METHOD M_User_SetAction : INT
VAR_INPUT
END_VAR
// TODO USER
//
// This method implements the logic for controlling a heater.
// There are two input values from sensors and two deltas for comparison.
//
// This example implements the heater control with the following assumptions:
//
// in_lrTemp1 - Lowest Temperature in the system (L)
// in_lrTemp2 - Temperature of the Detector (D). Coming from Lakeshore.
//
// The heater should keep the System temperature  
// in_lrPar1 to in_lrPar2 lower than the detector temperature.
// 
// in_lrPar1  - Delta [K] to turn the heater ON:  IF L < D - in_lrPar1
// in_lrPar2  - Delta [K] to turn the heater OFF: IF L > D - in_lrPar2
//
// in_lrDelta1 > in_lrDelta2, e.g. 10K > 4K.
//
// For example:
// 	in_lrPar1 = 10K
// 	in_lrPar1 = 4K
// 	Detector temperature D = 100K
// 	The lowest system temperature is kept in range [(100-10)..(100-4)] = [90K..96K].
//	The heater is turned ON  at < 90K.
//	The heater is turned OFF at > 96K.
//
IF	stat.nState = E_CRYO_BIN_CTRL_STATE.ACTIVE_OFF  OR  
	stat.nState = E_CRYO_BIN_CTRL_STATE.ACTIVE_ON THEN
	
	IF in_lrTemp1 < in_lrTemp2 - in_lrDelta_Low THEN
		// Activate the actuator
		M_User_SetAction	:= E_CRYO_BIN_CTRL_ACTION.ON;
	ELSIF in_lrTemp1 > in_lrTemp2 - in_lrDelta_High THEN
		// Dectivate the actuator
		M_User_SetAction	:= E_CRYO_BIN_CTRL_ACTION.OFF;
	END_IF

ELSE
	// Don't do anything
	M_User_SetAction	:= E_CRYO_BIN_CTRL_ACTION.NONE;
END_IF
END_METHOD

END_FUNCTION_BLOCK

// POUs/Actuators/FB_CRYO_LN2_CTRL
FUNCTION_BLOCK FB_CRYO_LN2_CTRL EXTENDS FB_CRYO_BIN_CTRL
VAR_INPUT
	in_lrTempK:		LREAL;			// Temperature input value [K]
	in_bValid:		BOOL := TRUE;	// Temperature Valid flag
	// Two parameters for decision making
	in_lrTempValveOpen:		LREAL := 91.27;		// Open  valve if temperature above this value [K]
	in_lrTempValveClose:	LREAL := 79.148;	// Close valve if temperature below this value [K]
END_VAR
VAR_OUTPUT
END_VAR
VAR
END_VAR

// Check the validity of the temperature reading.
// Start the check after 200 cycles.
IF stat.nCycleCounter > 200 THEN
	IF NOT in_bValid THEN
		// The temperature is not valid. 
		// The controller cannot work.
		stat.bCtrlOK	:= FALSE;
	ELSIF in_lrTempValveClose >= in_lrTempValveOpen THEN
		// Wrong configuration.
		// ValveClose MUST be lower than ValveOpen temperature
		stat.bCtrlOK	:= FALSE;
	ELSE
		// The temperature is valid. 
		stat.bCtrlOK	:= TRUE;
	END_IF
ELSE
	// The temperature is valid. 
	stat.bCtrlOK	:= TRUE;
END_IF

// Execute parent FB.
SUPER^();

METHOD M_SetStatus
VAR_INPUT
	nState:	E_CRYO_BIN_CTRL_STATE;
END_VAR
// Execute the status of the parent FB
SUPER^.M_SetStatus(nState);

// Set proper error description, if any.
IF Actuator.stat.bError THEN
	stat.sState	:= 'Valve failure';
ELSIF NOT stat.bCtrlOK THEN
	stat.sState	:= 'Temperature not valid';
END_IF
END_METHOD

METHOD M_User_SetAction : INT
VAR_INPUT
END_VAR
// TODO USER
// Overwrite Method FB_CRYO_BIN_CTRL::M_User_SetOutput()
//
// This method implements the logic for controlling the LN2 valve.
// 
// FB_CRYO_LN2_CTRL input parameters:
//
// in_lrTempK          - LN2 temperature
// in_bValid           - Flag if temperature reading is valid
// in_lrTempValveOpen  - Temperature upper limit [K]. Valve opens  when:  LN2 > in_lrTempValveOpen
// in_lrTempValveClose - Temperature lower limit [K]. Valve closes when:  LN2 < in_lrTempValveClose
//
// in_lrTempValveOpen > in_lrTempValveClose, e.g. 91.27K > 79.148K.
//
	
IF	stat.nState = E_CRYO_BIN_CTRL_STATE.ACTIVE_OFF  OR  
	stat.nState = E_CRYO_BIN_CTRL_STATE.ACTIVE_ON THEN
	// Check if input temperature value is valid.
	// If OK, check temperature against the limits	
	IF NOT stat.bCtrlOK THEN
		// Temperature reading is not valid.
		// Dectivate the actuator, i.e. close the valve
		M_User_SetAction	:= E_CRYO_BIN_CTRL_ACTION.OFF;
		stat.nState	:= E_CRYO_BIN_CTRL_STATE.ERROR;
	ELSIF in_lrTempK > in_lrTempValveOpen THEN
		// Activate the actuator, i.e. open the valve
		M_User_SetAction	:= E_CRYO_BIN_CTRL_ACTION.ON;
	ELSIF in_lrTempK < in_lrTempValveClose THEN
		// Dectivate the actuator, i.e. close the valve
		M_User_SetAction	:= E_CRYO_BIN_CTRL_ACTION.OFF;
	END_IF
	
ELSE
	// Don't do anything
	M_User_SetAction	:= E_CRYO_BIN_CTRL_ACTION.NONE;
END_IF
END_METHOD

END_FUNCTION_BLOCK

// POUs/Actuators/FB_CRYO_VALVE_CTRL
FUNCTION_BLOCK FB_CRYO_VALVE_CTRL EXTENDS FB_CRYO_BIN_CTRL
VAR_INPUT
END_VAR
VAR_OUTPUT
END_VAR
VAR
END_VAR

// Execute parent FB.
SUPER^();

METHOD M_SetStatus
VAR_INPUT
	nState:	E_CRYO_BIN_CTRL_STATE;
END_VAR
// Execute the status of the parent FB
SUPER^.M_SetStatus(nState);

// Set proper error description, if any.
IF Actuator.stat.bError THEN
	stat.sState	:= 'Valve failure';
END_IF
END_METHOD

METHOD M_User_SetAction : INT
VAR_INPUT
END_VAR
// TODO USER
// Set Valve command based on the input parameter in_bEnable.
//
	
IF	stat.nState = E_CRYO_BIN_CTRL_STATE.ACTIVE_OFF  AND in_bEnable THEN
	// Activate the actuator, i.e. open the valve
	M_User_SetAction	:= E_CRYO_BIN_CTRL_ACTION.ON;
ELSIF  stat.nState = E_CRYO_BIN_CTRL_STATE.ACTIVE_ON AND NOT in_bEnable THEN
	// Dectivate the actuator, i.e. close the valve
	M_User_SetAction	:= E_CRYO_BIN_CTRL_ACTION.OFF;
ELSE
	// Don't do anything
	M_User_SetAction	:= E_CRYO_BIN_CTRL_ACTION.NONE;
END_IF
END_METHOD

END_FUNCTION_BLOCK

// POUs/Comm/FB_MODBUS_COMM_CPA
FUNCTION_BLOCK FB_MODBUS_COMM_CPA EXTENDS FB_MODBUS_COMM_BASE
VAR_INPUT
END_VAR
VAR_OUTPUT
END_VAR
VAR CONSTANT
END_VAR
VAR
	{attribute 'OPC.UA.DA' := '0'}
	sim:		FB_SIM_MODBUS_COMM_CPA;	// Reference to COMM simulator

END_VAR

simRef	REF=sim;

// Execute base FB, i.e. FB_MODBUS_COMM_BASE.
SUPER^();

END_FUNCTION_BLOCK

// POUs/Simulation/FB_SIM_MODBUS_COMM_CPA
FUNCTION_BLOCK FB_SIM_MODBUS_COMM_CPA EXTENDS FB_SIM_MODBUS_COMM_BASE
VAR_INPUT
END_VAR
VAR_OUTPUT
END_VAR
VAR
END_VAR

M_ActivityDo();

METHOD M_GetSimReply : STRING(255)
VAR_INPUT
	{attribute 'OPC.UA.DA' := '0'}
	cmd:	STRING(16);		// MODBUS command. Only first 8 bytes are used
END_VAR
VAR
	sReply:		ARRAY [0..300] OF BYTE;
	sReply1:	STRING(255);
	n2Bytes:	ARRAY [0..1] OF BYTE;	// 2 bytes
	n4Bytes:	ARRAY [0..3] OF BYTE;	// 4 bytes
	i:			INT;
	nRegister:	INT;
	nWords:		INT;
	nPos:		INT;	
END_VAR
// TODO User: Implement simulator replies in FBs that EXTEND FB_SIM_MODBUS_COMM_BASE.
//            Only case where cmd[1] = E_MODBUS_CMD_TYPE.READ should be implemented.

IF cmd[1] = E_MODBUS_CMD_TYPE.WRITE THEN
// This is a WRITE command.
// Reply is the same as the command.
(*
	FOR i:=0 TO 8 DO
		sReply[i]	:= cmd[i];
	END_FOR
	*)
	M_GetSimReply := cmd;	
ELSE
// This is a READ command
	// Get register number - cmd[2..3] swapped bytes
	nRegister	:= M_ByteSwapINT(ADR(cmd[2]));

	// Get number of words - cmd[4..5] swapped bytes
	nWords	:= M_ByteSwapINT(ADR(cmd[4]));

	sReply[0]	:= cmd[0];
	sReply[1]	:= cmd[1];
	sReply[2]	:= INT_TO_BYTE(nWords * 2);
	
	IF nRegister = 16#0001 THEN		// common data
// nOperatingState
// 30,001 - Operating State
// 	3: stat.sOperatingState := 'Running';
// Offset 3 + 0x2 = 3
		nPos	:= 3;
		n2Bytes := M_ByteSwap_INT_TO_BYTES(3);
		M_InsertBytes_INT(s1:=sReply, s2:=n2Bytes, nPos:=nPos);

// nCompressorRunning
// 30,002 - Compressor Running == 1
// Offset 3 + 1x2 = 5
		nPos	:= 5;
		n2Bytes := M_ByteSwap_INT_TO_BYTES(1);
		M_InsertBytes_INT(s1:=sReply, s2:=n2Bytes, nPos:=nPos);

// nPos	:= nPos + 2;
// stat.lrWarningState := M_ByteSwapFLOAT(ADR(pBuf[nPos]));
		nPos	:= 7;
		n4Bytes := M_ByteSwap_REAL_TO_BYTES(0.0);
		M_InsertBytes_REAL(s1:=sReply, s2:=n4Bytes, nPos:=nPos);

// nPos	:= nPos + 4;
// stat.lrAlarmState := M_ByteSwapFLOAT(ADR(pBuf[nPos]));
		nPos	:= 11;
		n4Bytes := M_ByteSwap_REAL_TO_BYTES(0.0);
		M_InsertBytes_REAL(s1:=sReply, s2:=n4Bytes, nPos:=nPos);

// lrCoolantInTemp
// 30,007 - Coolant In Temp
// Offset 3 + 6x2 = 15
// nPos	:= nPos + 4;
// stat.lrCoolantInTemp	:= M_ByteSwapFLOAT(ADR(pBuf[nPos]));
		nPos	:= 15;
		n4Bytes := M_ByteSwap_REAL_TO_BYTES(M_GenerateRandom_REAL(17.0,1.0));
		M_InsertBytes_REAL(s1:=sReply, s2:=n4Bytes, nPos:=nPos);

// lrCoolantOutTemp
// 30,009 - Coolant Out Temp
// Offset 3 + 8x2 = 19
// nPos	:= nPos + 4;
// stat.lrCoolantOutTemp	:= M_ByteSwapFLOAT(ADR(pBuf[nPos]));
		nPos	:= 19;
		n4Bytes := M_ByteSwap_REAL_TO_BYTES(M_GenerateRandom_REAL(28.5,1.0));
		M_InsertBytes_REAL(s1:=sReply, s2:=n4Bytes, nPos:=nPos);

// lrOilTemp
// 30,011 - Oil Temp
// Offset 3 + 10x2 = 23
//nPos	:= nPos + 4;
//stat.lrOilTemp	:= M_ByteSwapFLOAT(ADR(pBuf[nPos]));
		nPos	:= 23;
		n4Bytes := M_ByteSwap_REAL_TO_BYTES(M_GenerateRandom_REAL(25.0,1.0));
		M_InsertBytes_REAL(s1:=sReply, s2:=n4Bytes, nPos:=nPos);

//nPos	:= nPos + 4;
//stat.lrHeliumTemp	:= M_ByteSwapFLOAT(ADR(pBuf[nPos]));
		nPos	:= 27;
		n4Bytes := M_ByteSwap_REAL_TO_BYTES(M_GenerateRandom_REAL(42.0,1.0));
		M_InsertBytes_REAL(s1:=sReply, s2:=n4Bytes, nPos:=nPos);


//nPos	:= nPos + 4;
//stat.lrLowPressure	:= M_ByteSwapFLOAT(ADR(pBuf[nPos]));
		nPos	:= 31;
		n4Bytes := M_ByteSwap_REAL_TO_BYTES(M_GenerateRandom_REAL(8.5,1.0));
		M_InsertBytes_REAL(s1:=sReply, s2:=n4Bytes, nPos:=nPos);

//nPos	:= nPos + 4;
//stat.lrLowPressureAverage	:= M_ByteSwapFLOAT(ADR(pBuf[nPos]));
		nPos	:= 35;
		n4Bytes := M_ByteSwap_REAL_TO_BYTES(M_GenerateRandom_REAL(8.5,1.0));
		M_InsertBytes_REAL(s1:=sReply, s2:=n4Bytes, nPos:=nPos);

//nPos	:= nPos + 4;
//stat.lrHighPressure	:= M_ByteSwapFLOAT(ADR(pBuf[nPos]));
		nPos	:= 39;
		n4Bytes := M_ByteSwap_REAL_TO_BYTES(M_GenerateRandom_REAL(21.0,1.0));
		M_InsertBytes_REAL(s1:=sReply, s2:=n4Bytes, nPos:=nPos);

//nPos	:= nPos + 4;
//stat.lrHighPressureAverage	:= M_ByteSwapFLOAT(ADR(pBuf[nPos]));
		nPos	:= 43;
		n4Bytes := M_ByteSwap_REAL_TO_BYTES(M_GenerateRandom_REAL(21.0,1.0));
		M_InsertBytes_REAL(s1:=sReply, s2:=n4Bytes, nPos:=nPos);

//nPos	:= nPos + 4;
//stat.lrDeltaPressureAverage	:= M_ByteSwapFLOAT(ADR(pBuf[nPos]));
		nPos	:= 47;
		n4Bytes := M_ByteSwap_REAL_TO_BYTES(M_GenerateRandom_REAL(12.0,1.0));
		M_InsertBytes_REAL(s1:=sReply, s2:=n4Bytes, nPos:=nPos);

//nPos	:= nPos + 4;
//stat.lrMotorCurrent	:= M_ByteSwapFLOAT(ADR(pBuf[nPos]));
		nPos	:= 51;
		n4Bytes := M_ByteSwap_REAL_TO_BYTES(M_GenerateRandom_REAL(12.1,0.09));
		M_InsertBytes_REAL(s1:=sReply, s2:=n4Bytes, nPos:=nPos);

//nPos	:= nPos + 4;
//stat.lrHoursOfOperation	:= M_ByteSwapFLOAT(ADR(pBuf[nPos]));
		nPos	:= 55;
		n4Bytes := M_ByteSwap_REAL_TO_BYTES(M_GenerateRandom_REAL(1633.3,0.0));
		M_InsertBytes_REAL(s1:=sReply, s2:=n4Bytes, nPos:=nPos);


//nPos	:= nPos + 4;
//stat.nPressureScale	:= M_ByteSwapINT(ADR(pBuf[nPos]));
		nPos	:= 59;
		n2Bytes := M_ByteSwap_INT_TO_BYTES(1);
		M_InsertBytes_INT(s1:=sReply, s2:=n2Bytes, nPos:=nPos);

//nPos	:= nPos + 2;
//stat.nTempScale	:= M_ByteSwapINT(ADR(pBuf[nPos]));
		nPos	:= 61;
		n2Bytes := M_ByteSwap_INT_TO_BYTES(1);
		M_InsertBytes_INT(s1:=sReply, s2:=n2Bytes, nPos:=nPos);

//nPos	:= nPos + 2;
//pPtr	:= ADR(pBuf[nPos]);
//stat.nPanelSerialNumber	:= pPtr^;
		nPos	:= 63;
		n2Bytes := M_ByteSwap_UINT_TO_BYTES(50464);
		M_InsertBytes_INT(s1:=sReply, s2:=n2Bytes, nPos:=nPos);

//nPos	:= nPos + 2;
//stat.nModelMajorMinor	:= M_ByteSwapINT(ADR(pBuf[nPos]));
		nPos	:= 65;
		n2Bytes := M_ByteSwap_INT_TO_BYTES(539);
		M_InsertBytes_INT(s1:=sReply, s2:=n2Bytes, nPos:=nPos);

	END_IF


	// TODO
	// Calculate CRC for the first 6 bytes
	//	crc	:= M_CRC(ADR(cmd),6);
	
	FOR i:=0 TO 254 DO
		sReply1[i]	:= sReply[i];
	END_FOR

	M_GetSimReply := sReply1;
END_IF
END_METHOD

END_FUNCTION_BLOCK

// POUs/Coolers/FB_CRYO_CPA
FUNCTION_BLOCK FB_CRYO_CPA EXTENDS FB_RS_BASE
VAR_INPUT
	{attribute 'OPC.UA.DA' := '0'}
	in_sSN_Compressor:	STRING;	// e.g. 'CPA289C-W2EHCE-180201A'
	{attribute 'OPC.UA.DA' := '0'}
	in_sSN_PulseTube:	STRING;	// e.g. 'CH40810-180208A'
	{attribute 'OPC.UA.DA' := '0'}
	in_nYear_Compressor:	INT;	// e.g. 2018
	{attribute 'OPC.UA.DA' := '0'}
	in_nYear_PulseTube:		INT;	// e.g. 2018
	{attribute 'OPC.UA.DA' := '0'}
	in_lrNextService_Compressor:	LREAL;	// Next service in absolute hours
	{attribute 'OPC.UA.DA' := '0'}
	in_lrNextService_PulseTube:		LREAL;	// Next service in absolute hours
	{attribute 'OPC.UA.DA' := '0'}
	in_nSlaveID:	BYTE := 1;		// Modbus Slave ID
	{attribute 'OPC.UA.DA' := '0'}
	in_nPeriod:		DINT := 5000;	//Interval for periodic reading [ms], default 5000 ms = 5 sec
END_VAR
VAR_OUTPUT
END_VAR
VAR CONSTANT
END_VAR
VAR
	{attribute 'OPC.UA.DA' := '1'}
	cfg:		T_CRYO_CPA_CFG;					//  Config parameters
	{attribute 'OPC.UA.DA' := '1'}
	ctrl:		T_CRYO_CPA_CTRL;				//  Control parameters
	{attribute 'OPC.UA.DA' := '1'}
	{attribute 'OPC.UA.DA.Access' := '1'}
	info:		T_CRYO_CPA_INFO; 				//  Info parameters - ReadOnly
	{attribute 'OPC.UA.DA' := '1'}
	{attribute 'OPC.UA.DA.Access' := '1'}
	stat:		T_CRYO_CPA_STAT;				//  Status parameters - ReadOnly

	{attribute 'OPC.UA.DA' := '0'}
	comm:		FB_MODBUS_COMM_CPA;				// Instance of generic comm object. OPC UA Disabled!!!
	
	(* Pointers *)
	{attribute 'OPC.UA.DA' := '0'}
	ptrCommCtrl:	POINTER TO T_MODBUS_CTRL 	:= ADR(comm.ctrl);	(* Pointer to comm.ctrl instance *)

	// I/O
	q_bCtrlStart	AT %Q*:	BOOL;	// Start control signal
	
	
	(* Timers *)
	{attribute 'OPC.UA.DA' := '0'}
	fbTimer:			TON; (* General Timeout *)
	
	// Dummy variables for testing
	nDummyWarnings:	DINT := 0;
	nDummyErrors:	DINT := 0;

END_VAR

// Set references
cfgRef	REF=cfg;
ctrlRef	REF=ctrl;
statRef	REF=stat;


// 
// Execute comm instance.
// Function 4 is used for READ.
//
comm(	in_bSimulation		:= in_bSimulation,
		in_cReadFunction	:= 4);


// Execute the base class object FB_RS_BASE
SUPER^();

METHOD ActivityInitializing
VAR_INPUT
	bExecute:	BOOL;
END_VAR
VAR_INST
	{attribute 'OPC.UA.DA' := '0'}
    nMethodState:	INT := 0;	// State Machine current state
END_VAR
VAR
	nInt:	INT;	// Temporary INT for conversion of ENUM types
END_VAR
SetAction('ActivityInitializing');


IF NOT bExecute THEN
	nMethodState	:= 0;	// Reset the state machine
	RETURN;
END_IF

// Handle State Machine
CASE nMethodState OF
	0:	// Set monitoring period (from input parameter)
		cfg.tDelay_Periodic	:= DINT_TO_TIME(in_nPeriod);
		// Auto monitor, i.e. monitor in Standby_Ready as well
		cfg.bAutoMonitor	:= TRUE;

		(* Set initial state and status *)
		stat.bInitialised	:= FALSE;
		stat.nRetries		:= 0;

		SetStatus(E_SM_ERROR.OK, 'BUSY');
		
		// User configuration of the system
		M_UserConfigure();

		nMethodState := 10;				// Go to next state, i.e. INIT_COMM

	10:	// Initialize COMM port, i.e. Reset the serial port.
		nInt	:= E_RS_COMM_CMD.INIT;
		ptrCommCtrl^.nCommand	:= nInt;
		ptrCommCtrl^.bExecute	:= TRUE;

		(* Start the timer by going false/true *)
		fbTimer (IN := FALSE); (* Reset timer *)
		fbTimer (IN := TRUE, PT := T#5S); (* 5 sec timeout for reply *)

		nMethodState := 15;	// On next cycle wait until comm port is reset, i.e. idle
		
	15:	// Wait IDLE or ERROR
		fbTimer (IN := TRUE);
		IF comm.stat.nStatus = E_RS_COMM_STATUS.IDLE THEN
			// Communication is IDLE 
			fbTimer (IN := FALSE);	// disable timer 
			stat.nInputBuffer		:= comm.stat.DeviceReply;	// Save the reply

			bCommProblem	:= FALSE;
			// Device INIT is done.
			// INITDONE will bring it to OPERATIONAL
			stat.bInitialised 	:= TRUE;
			SetStatus(E_CCC_STATUS.IDLE, 'IDLE');
			nEvent 	:= E_SM_EVENT.INITDONE;
			RETURN;
		ELSIF comm.stat.nStatus = E_RS_COMM_STATUS.ERROR OR fbTimer.Q THEN
			// There is an error.
			// Re-initialise the comm port.
			// This is the only thing we can do.
			SetStatus(E_CCC_ERROR.COMM, 'ERROR: Communication error');	
			bCommProblem	:= TRUE;
			nMethodState	:= 10;		// Retry to INIT_COMM
			RETURN;
		END_IF
	
END_CASE
END_METHOD

METHOD ActivityMonitoring
VAR_INPUT
	bExecute:	BOOL;
END_VAR
VAR_INST
	{attribute 'OPC.UA.DA' := '0'}
    nMethodState:	INT := 0;					// State Machine current state
	{attribute 'OPC.UA.DA' := '0'}
	nSlaveIndex:	INT := 1;
	{attribute 'OPC.UA.DA' := '0'}
	nRetries:		INT := 0;					// Number of retries in case of communication problems
END_VAR
IF NOT bExecute THEN
	SetAction('ActivityMonitoring'); 
	SetStatus(E_SM_ERROR.OK, 'BUSY');
	nMethodState	:= 0;	// Reset the state machine
	ctrl.nSlaveID	:= cfg.nSlaveID;
	ctrl.nRegister	:= cfg.nAddrCommon;
	ctrl.nWords		:= cfg.nWordsCommon;
	nRetries		:= 0;					
	RETURN;
END_IF

// Handle State Machine
CASE nMethodState OF
	0:	// Execute a command from the command array
		// Check if we have to exit Monitoring
		
		// Send command
		ptrCommCtrl^.nCommand	:= E_MODBUS_CMD.SEND;
		ptrCommCtrl^.nSlaveID	:= ctrl.nSlaveID;
		ptrCommCtrl^.nRegister	:= ctrl.nRegister;
		ptrCommCtrl^.nWords		:= ctrl.nWords;
		ptrCommCtrl^.bExecute	:= TRUE;
		
		(* Start the timer by going false/true *)
		fbTimer (IN := FALSE); (* Reset timer *)
		fbTimer (IN := TRUE, PT := T#5S); (* 5 sec timeout for reply *)

		nMethodState := 20;				// Goto WAIT for Reading to complete,

	10:	// Wait until the delay timeout expires
		fbTimer (IN := TRUE);

		(* If Timer has expired, go to the next state. *)
		IF fbTimer.Q THEN
			fbTimer (IN := FALSE);
			SetStatus(E_SM_ERROR.OK, 'BUSY');
			nMethodState 	:= 0;	// Goto next reading
			RETURN;
		END_IF
	


	20:	// Wait for the reading to complete, i.e. IDLE
		fbTimer (IN := TRUE);
		IF comm.stat.nStatus = E_RS_COMM_STATUS.IDLE THEN
			//
			// Communication is IDLE. Everything is fine. 
			//
			fbTimer (IN := FALSE);	// disable timer 
			stat.nInputBuffer	:= comm.stat.DeviceReply;	// Save the reply
			
			//
			// Extract the readings from the reply.
			//
			M_ExtractReadings();
			
			bCommProblem	:= FALSE;
			nRetries		:= 0;	// Reset number of retries
			
			// Wait tDelay_Periodic before re-starting the READ.
			SetStatus(E_SM_ERROR.OK, 'IDLE');
			(* Start the timer by going false/true *)
			fbTimer (IN := FALSE); (* Reset timer *)
			fbTimer (IN := TRUE, PT := cfg.tDelay_Periodic);
			nMethodState := 10;				// Goto Wait 
			RETURN;

		ELSIF INT_TO_DINT(comm.stat.nStatus) = INT_TO_DINT(E_MODBUS_STATUS.ERROR) OR fbTimer.Q THEN
			//
			// There is a communication problem. 
			// Re-initialise comm port.
			//
			fbTimer (IN := FALSE);
			SetStatus(E_MODBUS_ERROR.RECEIVE, 'ERROR: Communication error');	
			bCommProblem	:= TRUE;
			
			// Keep track of how many times we re-tried
			nRetries		:= nRetries + 1;		// Increment number of retries
			stat.nRetries	:= stat.nRetries + 1;	// Increment total number of retries

			// Re-initialise the comm port
			ptrCommCtrl^.nCommand	:= E_MODBUS_CMD.INIT;
			ptrCommCtrl^.bExecute	:= TRUE;
			// Apply a delay of 3 sec and retry
			fbTimer (IN := FALSE); (* Reset timer *)
			fbTimer (IN := TRUE, PT := T#3000MS);
			nMethodState := 10;				// Goto Wait 
			RETURN;
		END_IF

	
END_CASE
END_METHOD

METHOD CheckForEvents
VAR_INPUT
END_VAR
VAR
//	nInt2:	INT;	// Temporary INT for conversion of ENUM types
END_VAR

(* 
	Check for events in the following order: 
   	1) HW failure: without HW avilability there is no point to do anything
	2) Internal events: to allow completing the initiated commands before 
                        starting processing new commands. 
   	3) Commands: to react to external commands. Commands should be executed 
                 before processing HW signals to allow to start a recovery action.
   	4) HW signals: if any.
*)

IF NOT M_GetCouplerState() THEN	
	(* Check if the HW is NOT OK *)
	(*
	If the hardware status is NOT OK, we cannot trust the readings.
	Variable i_nCouplerState has to be mapped to a State of a terminal, e.g. EK1100.
	The value should be 8.
 	*)
	SetEvent(E_SM_EVENT.ERRHW);
	SetStatus(E_SM_ERROR.HW_NOT_OP, 'ERROR: HW not in OPERATIONAL state');

ELSIF ctrlRef.bExecute  THEN
	// Check for CPA specific commands.
	// TODO SetLastCommand() and SetEvent() don't work here. Check it!!!
	ctrlRef.bExecute	:= FALSE;			(* Clear the Execute bit *)
	SetLastCommand(E_RS_COMMAND.CTRL_CMD);	// Save the last command
	SetEvent(E_RS_COMMAND.CTRL_CMD);
	IF	ctrl.nDevCommand = E_CRYO_CPA_CMDS.START	THEN
		// Set control signal to TRUE.
		// This will start the compressor.
		q_bCtrlStart	:= TRUE;
	ELSIF	ctrl.nDevCommand = E_CRYO_CPA_CMDS.STOP	THEN
		// Set control signal to FALSE.
		// This will stop the compressor.
		q_bCtrlStart	:= FALSE;
	ELSE
		(* Handle standard RS commands *)
		SetLastCommand(ctrlRef.nCommand);			(* Save the last command *)
		SetEvent(ctrlRef.nCommand);
	END_IF
	ctrlRef.bExecute	:= FALSE;			(* Clear the Execute bit *)
	ctrlRef.nCommand 	:= E_RS_COMMAND.NONE;	(* Clear the Command *)
ELSIF nInternalEvent <> E_SM_EVENT.NONE THEN
	(* Handle internal events *)
	SetEvent(nInternalEvent);
	nInternalEvent := E_SM_EVENT.NONE;
ELSE
	(* Handle HW problems and unexpected bahaviour *)
	
END_IF
END_METHOD

METHOD M_ByteSwapFLOAT : LREAL
VAR_INPUT
	pByte:		POINTER TO BYTE;	// Pointer to array of bytes read from JUMO
END_VAR
VAR
	rResult:	REAL;
	pResult:	POINTER TO BYTE	:= ADR(rResult);	// Pointer to the result
END_VAR
pResult[0]	:= pByte[1];
pResult[1]	:= pByte[0];
pResult[2]	:= pByte[3];
pResult[3]	:= pByte[2];

M_ByteSwapFLOAT	:= REAL_TO_LREAL(rResult);
END_METHOD

METHOD M_ByteSwapINT : INT
VAR_INPUT
	pByte:		POINTER TO BYTE;	// Pointer to array of bytes read from JUMO
END_VAR
VAR
	nResult:	INT;
	pResult:	POINTER TO BYTE	:= ADR(nResult);	// Pointer to the result
END_VAR
pResult[0]	:= pByte[1];
pResult[1]	:= pByte[0];

M_ByteSwapINT	:= nResult;
END_METHOD

METHOD M_CheckDiagnostics
VAR_INPUT
END_VAR
VAR
	nTmp:		DINT;
	i:			INT;
	sTmp:		STRING(56) := '';
END_VAR
// Process warnings/alarms
//M_CheckWarnings(stat.lrWarningState);
M_CheckWarnings(nDummyWarnings);

// Process errors
//M_CheckErrors(stat.lrWarningState);
M_CheckErrors(nDummyErrors);
END_METHOD

METHOD M_CheckErrors
VAR_INPUT
	nErrors:	DINT;
END_VAR
VAR
	nTmp:		UDINT;
	nRef:		UDINT	:= 16#00000001;
	bProblem:	BOOL	:= FALSE;
	i:			INT;
END_VAR
nTmp	:= DINT_TO_UDINT(-nErrors);


FOR i := 0 TO 6 DO
	// Check for 'too low' errors
	IF		(stat.aReadings[i] < cfg.aLimits[i].rErrorLow) OR
			((nTmp AND SHL(nRef,cfg.aDiag[i].nBitLow)) <> 0)	THEN
		bProblem	:= TRUE;
		stat.arrErrors[i]		:= E_CRYO_CPA_ALARM.LOW;
		M_SetAlarmText(i);	// Error string for going low
	// Check for 'too high' errors
	ELSIF	(stat.aReadings[i] > cfg.aLimits[i].rErrorHigh) OR
			((nTmp AND SHL(nRef,cfg.aDiag[i].nBitHigh)) <> 0)	THEN
		bProblem	:= TRUE;
		stat.arrErrors[i]		:= E_CRYO_CPA_ALARM.HIGH;
		M_SetAlarmText(i);	// Error string for going high
	ELSE
		stat.arrErrors[i]	:= E_CRYO_CPA_ALARM.NONE;
	END_IF
END_FOR

// Check if there are any errors.
IF NOT bProblem THEN
	// No error. Clear all and write OK in warning text.
	FOR i := 0 TO 6 DO
		stat.arrErrors[i]	:= E_CRYO_CPA_ALARM.NONE;
	END_FOR
	stat.sError := '';
//  We don't touch stat.nStatusCode! It might have been set with alarm.
	RETURN;
ELSE
	stat.nStatusCode	:= 2;	// Error
END_IF
END_METHOD

METHOD M_CheckService
VAR_INPUT
END_VAR
VAR
    fbFormat: FB_FormatString;
	lrHoursLeft:	LREAL;
END_VAR
//
// Check compressor hours
//
lrHoursLeft	:= in_lrNextService_Compressor - stat.lrHoursOfOperation;
IF lrHoursLeft < cfg.lrServiceDue_Compressor THEN
	stat.bServiceDue_Compressor	:= TRUE;
	stat.wColour_Compressor		:= 16#FFFF0000;
	IF lrHoursLeft >= 0.0 THEN
		fbFormat( 	sFormat := 'Service due in %.0f hours', 
					arg1 := F_LREAL( lrHoursLeft ), 
					sOut => stat.sServiceDue_Compressor);
	ELSE
		lrHoursLeft	:= -1 * lrHoursLeft;
		fbFormat( 	sFormat := 'Service overdue by %.0f hours', 
					arg1 := F_LREAL( lrHoursLeft ), 
					sOut => stat.sServiceDue_Compressor);
	END_IF
ELSE
	stat.wColour_Compressor		:= 16#FF0000FF;
	stat.bServiceDue_Compressor	:= FALSE;
	stat.sServiceDue_Compressor	:= 'OK';
END_IF

//
// Check pulse tube hours
//
lrHoursLeft	:= in_lrNextService_PulseTube - stat.lrHoursOfOperation;
IF lrHoursLeft < cfg.lrServiceDue_PulseTube THEN
	stat.bServiceDue_PulseTube	:= TRUE;
	stat.wColour_PulseTube		:= 16#FFFF0000;
	IF lrHoursLeft >= 0.0 THEN
		fbFormat( 	sFormat := 'Service due in %.0f hours', 
					arg1 := F_LREAL( lrHoursLeft ), 
					sOut => stat.sServiceDue_PulseTube);
	ELSE
		lrHoursLeft	:= -1 * lrHoursLeft;
		fbFormat( 	sFormat := 'Service overdue by %.0f hours', 
					arg1 := F_LREAL( lrHoursLeft ), 
					sOut => stat.sServiceDue_PulseTube);
	END_IF
ELSE
	stat.wColour_PulseTube		:= 16#FF0000FF;
	stat.bServiceDue_PulseTube	:= FALSE;
	stat.sServiceDue_PulseTube	:= 'OK';
END_IF
END_METHOD

METHOD M_CheckWarnings
VAR_INPUT
	nWarnings:	DINT;
END_VAR
VAR
	nTmp:		UDINT;
	nRef:		UDINT	:= 16#00000001;
	bProblem:	BOOL	:= FALSE;
	i:			INT;
END_VAR
// Warning are given as negative numbers.
// Change the sign and then do checks with bit shifts to the left.
nTmp	:= DINT_TO_UDINT(-nWarnings);

// Check warnings one by one
FOR i := 0 TO 6 DO
	// Check for 'running low' warnings/alarms
	IF		(stat.aReadings[i] < cfg.aLimits[i].rAlarmLow) OR
			((nTmp AND SHL(nRef,cfg.aDiag[i].nBitLow)) <> 0)	THEN
		bProblem	:= TRUE;
		stat.arrAlarms[i]		:= E_CRYO_CPA_ALARM.LOW;
		M_SetAlarmText(i);	// Alarm string for going low (FALSE)
	// Check for 'running high' warnings/alarms
	ELSIF	(stat.aReadings[i] > cfg.aLimits[i].rAlarmHigh) OR
			((nTmp AND SHL(nRef,cfg.aDiag[i].nBitHigh)) <> 0)		THEN
		bProblem	:= TRUE;
		stat.arrAlarms[i]		:= E_CRYO_CPA_ALARM.HIGH;
		M_SetAlarmText(i);	// Alarm string for going high (TRUE)
	ELSE
		stat.arrAlarms[i]	:= E_CRYO_CPA_ALARM.NONE;
	END_IF
END_FOR

// Check if there are any alarms.
IF NOT bProblem THEN
	// No alarms. Clear all and write OK in warning text.
	FOR i := 0 TO 6 DO
		stat.arrAlarms[i]	:= E_CRYO_CPA_ALARM.NONE;
	END_FOR
	stat.sAlarm := '';
	stat.nStatusCode	:= 0;	// OK
ELSE
	stat.nStatusCode	:= 1;	// Alarm
END_IF
END_METHOD

METHOD M_ExtractReadings : BOOL
VAR_INPUT
END_VAR
VAR
	pBuf:	POINTER TO BYTE	:= ADR(stat.nInputBuffer);
	nPos:	INT	:= 0;	// byte position in the buffer
	pPtr:	POINTER TO UINT;	// Pointer to the result
END_VAR
// There are 3 bytes before data starts !!!
////////////////////////////
// Extract Common Parameters
// Buffer starts from 30,001
// 3 bytes before real data
////////////////////////////

// nOperatingState
// 30,001 - Operating State
// Offset 3 + 0x2 = 3
nPos	:= cfg.nPosOffset + 3;
stat.nOperatingState := M_ByteSwapINT(ADR(pBuf[nPos]));

// nCompressorRunning
// 30,002 - Compressor Running
// Offset 3 + 1x2 = 5
nPos	:= nPos + 2;
stat.nCompressorRunning := M_ByteSwapINT(ADR(pBuf[nPos]));

// 
// 
// Offset 3 + x2 = 
nPos	:= nPos + 2;
stat.lrWarningState := M_ByteSwapFLOAT(ADR(pBuf[nPos]));

// 
// 
// Offset 3 + x2 = 
nPos	:= nPos + 4;
stat.lrAlarmState := M_ByteSwapFLOAT(ADR(pBuf[nPos]));

// lrCoolantInTemp
// 30,007 - Coolant In Temp
// Offset 3 + 6x2 = 15
nPos	:= nPos + 4;
stat.lrCoolantInTemp	:= M_ByteSwapFLOAT(ADR(pBuf[nPos]));

// lrCoolantOutTemp
// 30,009 - Coolant Out Temp
// Offset 3 + 8x2 = 19
nPos	:= nPos + 4;
stat.lrCoolantOutTemp	:= M_ByteSwapFLOAT(ADR(pBuf[nPos]));

// lrOilTemp
// 30,011 - Oil Temp
// Offset 3 + 10x2 = 23
nPos	:= nPos + 4;
stat.lrOilTemp	:= M_ByteSwapFLOAT(ADR(pBuf[nPos]));

nPos	:= nPos + 4;
stat.lrHeliumTemp	:= M_ByteSwapFLOAT(ADR(pBuf[nPos]));

nPos	:= nPos + 4;
stat.lrLowPressure	:= M_ByteSwapFLOAT(ADR(pBuf[nPos]));

nPos	:= nPos + 4;
stat.lrLowPressureAverage	:= M_ByteSwapFLOAT(ADR(pBuf[nPos]));

nPos	:= nPos + 4;
stat.lrHighPressure	:= M_ByteSwapFLOAT(ADR(pBuf[nPos]));

nPos	:= nPos + 4;
stat.lrHighPressureAverage	:= M_ByteSwapFLOAT(ADR(pBuf[nPos]));

nPos	:= nPos + 4;
stat.lrDeltaPressureAverage	:= M_ByteSwapFLOAT(ADR(pBuf[nPos]));

nPos	:= nPos + 4;
stat.lrMotorCurrent	:= M_ByteSwapFLOAT(ADR(pBuf[nPos]));

nPos	:= nPos + 4;
stat.lrHoursOfOperation	:= M_ByteSwapFLOAT(ADR(pBuf[nPos]));

nPos	:= nPos + 4;
stat.nPressureScale	:= M_ByteSwapINT(ADR(pBuf[nPos]));

nPos	:= nPos + 2;
stat.nTempScale	:= M_ByteSwapINT(ADR(pBuf[nPos]));

nPos	:= nPos + 2;
pPtr	:= ADR(pBuf[nPos]);
stat.nPanelSerialNumber	:= pPtr^;
//stat.nPanelSerialNumber	:= M_ByteSwapINT(ADR(pBuf[nPos]));

nPos	:= nPos + 2;
stat.nModelMajorMinor	:= M_ByteSwapINT(ADR(pBuf[nPos]));

//////////////////////////
// Assign values to arrays
//////////////////////////

stat.aReadings[E_CRYO_CPA_DIAG_IDX.WATER_IN]	:= stat.lrCoolantInTemp;
stat.aReadings[E_CRYO_CPA_DIAG_IDX.WATER_OUT]	:= stat.lrCoolantOutTemp;
stat.aReadings[E_CRYO_CPA_DIAG_IDX.OIL_TEMP]	:= stat.lrOilTemp;
stat.aReadings[E_CRYO_CPA_DIAG_IDX.HELIUM_TEMP]	:= stat.lrHeliumTemp;
stat.aReadings[E_CRYO_CPA_DIAG_IDX.HELIUM_LOW_PRESS_OP]		:= stat.lrLowPressure;
stat.aReadings[E_CRYO_CPA_DIAG_IDX.HELIUM_HIGH_PRESS_OP]	:= stat.lrHighPressure;

IF stat.nCompressorRunning <> 0 THEN
	stat.bSystemOn	:= TRUE;
	cfg.aLimits	:= cfg.aLimits_OP;
	
	// System is ON. Set 'operational' values to the actual reading.
	stat.aReadings[E_CRYO_CPA_DIAG_IDX.HELIUM_DELTA_PRESS]		:= stat.lrDeltaPressureAverage;
ELSE
	stat.bSystemOn	:= FALSE;
	cfg.aLimits	:= cfg.aLimits_ST;
	
	// System is OFF. 
	// Set 'static' values to the middle of the valid range to avoid warnings and errors.
	stat.aReadings[E_CRYO_CPA_DIAG_IDX.HELIUM_DELTA_PRESS]		:= 12.0;	// dummy
END_IF

//
// Check for Alarms and Errors
//
M_CheckDiagnostics();

//
// Get Model Number
//
M_GetModelNumber();

//
// Get Operational State
//
M_GetOperatingState();

//
// Check due service
//
M_CheckService();
END_METHOD

METHOD M_GetModelNumber
VAR_INPUT
END_VAR
VAR
	nModelMajor:	SINT;
	nModelMinor:	SINT;
	nVersionMajor:	SINT;
	nVersionMinor:	SINT;
	pPtr:			POINTER TO BYTE;;	// Pointer to the result
	sModelMajor, sModelMinor:	STRING(16);
	sVersionMajor, sVersionMinor:	STRING(16);
	sTmp:	STRING;
END_VAR
// Get major and minor version of the model
pPtr	:= ADR(stat.nModelMajorMinor);
nModelMinor	:= BYTE_TO_SINT(pPtr^);

pPtr	:= ADR(stat.nModelMajorMinor) + 1;
nModelMajor	:= BYTE_TO_SINT(pPtr^);

CASE nModelMajor OF
	1:	sModelMajor	:= '8';
	2:	sModelMajor	:= '9';
	3:	sModelMajor	:= '10';
	4:	sModelMajor	:= '11';
	5:	sModelMajor	:= '28';
END_CASE

CASE nModelMinor OF
	1:	sModelMinor	:= 'A1';
	2:	sModelMinor	:= '01';
	3:	sModelMinor	:= '02';
	4:	sModelMinor	:= '03';
	5:	sModelMinor	:= 'H3';
	6:	sModelMinor	:= 'I3';
	7:	sModelMinor	:= '04';
	8:	sModelMinor	:= 'H4';
	9:	sModelMinor	:= '05';
	10:	sModelMinor	:= 'H5';
	11:	sModelMinor	:= 'I6';
	12:	sModelMinor	:= '06';
	13:	sModelMinor	:= '07';
	14:	sModelMinor	:= 'H7';
	15:	sModelMinor	:= 'I7';
	16:	sModelMinor	:= '08';
	17:	sModelMinor	:= '09';
	18:	sModelMinor	:= '9C';
	19:	sModelMinor	:= '10';
	20:	sModelMinor	:= '1I';
	21:	sModelMinor	:= '11';
	22:	sModelMinor	:= '12';
	23:	sModelMinor	:= '13';
	24:	sModelMinor	:= '14';
END_CASE

// Get major and minor version of the panel
pPtr	:= ADR(stat.nPanelSerialNumber);
nVersionMinor	:= BYTE_TO_SINT(pPtr^);

pPtr	:= ADR(stat.nPanelSerialNumber) + 1;
nVersionMajor	:= BYTE_TO_SINT(pPtr^);


sTmp	:= 'CRYOMECH CPA';
sTmp	:= concat(concat(sTmp,sModelMajor),sModelMinor);
sTmp	:= concat(concat(sTmp,'   ID: '),in_sName);
//sTmp	:= concat(concat(sTmp,'.'),SINT_TO_STRING(nVersionMinor));

stat.sModelNumber	:= sTmp;



(*
Major Model Numbers consist of
1: 800 Series
2: 900 Series
3: 1000 Series
4: 1100 Series
5: 2800 Series
Minor Model Numbers consist of:
1: A1 13: 07
2: 01 14: H7
3: 02 15: I7
4: 03 16: 08
5: H3 17: 09
6: I3 18: 9C
7: 04 19: 10
8: H4 20: 1I
9: 05 21: 11
10: H5 22: 12
11: I6 23: 13
12: 06 24: 14
*)
END_METHOD

METHOD M_GetOperatingState
VAR_INPUT
END_VAR

VAR
	
END_VAR
CASE stat.nOperatingState OF
	0: stat.sOperatingState := 'Idling - ready to start';
	2: stat.sOperatingState := 'Starting';
	3: stat.sOperatingState := 'Running';
	5: stat.sOperatingState := 'Stopping';
	6: stat.sOperatingState := 'Error Lockout';
	7: stat.sOperatingState := 'Error';
	8: stat.sOperatingState := 'Helium Cool Down';
	9: stat.sOperatingState := 'Error-Power Related';
	16: stat.sOperatingState := 'Error Recovery';
END_CASE




(*
Input Register 30001: (operating state)
0: Idling - ready to start
2: Starting
3: Running
5: Stopping
6: Error Lockout
7: Error
8: Helium Cool Down
9: Error-Power Related
16: Error Recovery
*)
END_METHOD

METHOD M_SetAlarmText
VAR_INPUT
	nIndex:	INT;	// alarm index
END_VAR
VAR
	sTmp1:	STRING(128);
END_VAR
//
// Handle alarms
//
IF stat.arrAlarms[nIndex] = E_CRYO_CPA_ALARM.NONE THEN
	// No alarm 
	stat.sAlarm	:= '';
ELSIF stat.arrAlarms[nIndex] = E_CRYO_CPA_ALARM.LOW THEN
	// Alarm text, e.g. 
	// ‘Alarm: High pressure running low, compressor will shut off at 27.6 bar’
	sTmp1	:= concat('Alarm: ', cfg.aDiag[nIndex].sLabel);
	sTmp1	:= concat(sTmp1, ' running low. It will shut down at ');
	sTmp1	:= concat(sTmp1, LREAL_TO_STRING(cfg.aDiag[nIndex].rErrorLow));
	sTmp1	:= concat(sTmp1, concat(' ', cfg.aDiag[nIndex].sUnits));
	stat.sAlarm	:= sTmp1;
ELSIF stat.arrAlarms[nIndex] = E_CRYO_CPA_ALARM.HIGH THEN
	// Alarm text, e.g. 
	// ‘Alarm: High pressure running high, compressor will shut off at 27.6 bar’
	sTmp1	:= concat('Alarm: ', cfg.aDiag[nIndex].sLabel);
	sTmp1	:= concat(sTmp1, ' running high. It will shut down at ');
	sTmp1	:= concat(sTmp1, LREAL_TO_STRING(cfg.aDiag[nIndex].rErrorHigh));
	sTmp1	:= concat(sTmp1, concat(' ', cfg.aDiag[nIndex].sUnits));
	stat.sAlarm	:= sTmp1;
END_IF

//
// Handle errors
//
IF stat.arrErrors[nIndex] = E_CRYO_CPA_ALARM.NONE THEN
	// No error 
	stat.sError	:= '';
ELSIF stat.arrErrors[nIndex] = E_CRYO_CPA_ALARM.LOW THEN
	// Error text, e.g. 
	// ‘Error: High pressure was too low, compressor shut down at 27.6 bar’
	sTmp1	:= concat('Error: ', cfg.aDiag[nIndex].sLabel);
	sTmp1	:= concat(sTmp1, ' was too low. Shutdown was at ');
	sTmp1	:= concat(sTmp1, LREAL_TO_STRING(cfg.aDiag[nIndex].rErrorLow));
	sTmp1	:= concat(sTmp1, concat(' ', cfg.aDiag[nIndex].sUnits));
	stat.sError	:= sTmp1;
ELSIF stat.arrErrors[nIndex] = E_CRYO_CPA_ALARM.HIGH THEN
	// Error text, e.g. 
	// ‘Error: High pressure was too high, compressor shut down at 27.6 bar’
	sTmp1	:= concat('Error: ', cfg.aDiag[nIndex].sLabel);
	sTmp1	:= concat(sTmp1, ' was too high. Shutdown was at ');
	sTmp1	:= concat(sTmp1, LREAL_TO_STRING(cfg.aDiag[nIndex].rErrorHigh));
	sTmp1	:= concat(sTmp1, concat(' ', cfg.aDiag[nIndex].sUnits));
	stat.sError	:= sTmp1;
END_IF
END_METHOD

METHOD M_UserConfigure : BOOL
VAR_INPUT
END_VAR
VAR
	i, j:	int;
END_VAR
// TODO USER
// Add here real configuration

// SlaveID
cfg.nSlaveID	:= in_nSlaveID;

// We always read from CPA
ctrl.nCmdType	:= E_MODBUS_CMD_TYPE.READ;

ctrl.nRegister	:= cfg.nAddrCommon;
ctrl.nWords		:= cfg.nWordsCommon;

//
// Configure OP and STATIC limits
FOR i := 0 TO 6 DO
	cfg.aLimits_OP[i].rAlarmLow	:= MAX(cfg.aDiag[i].rAlarmLow_CPA,  cfg.aDiag[i].rAlarmLow_ESO);
	cfg.aLimits_OP[i].rAlarmHigh	:= MIN(cfg.aDiag[i].rAlarmHigh_CPA, cfg.aDiag[i].rAlarmHigh_ESO);
	cfg.aLimits_OP[i].rErrorLow	:= cfg.aDiag[i].rErrorLow;
	cfg.aLimits_OP[i].rErrorHigh	:= cfg.aDiag[i].rErrorHigh;

	j	:= i;
	IF	i = E_CRYO_CPA_DIAG_IDX.HELIUM_LOW_PRESS_OP OR 
		i = E_CRYO_CPA_DIAG_IDX.HELIUM_HIGH_PRESS_OP THEN
		j	:= i+3;	// Use STATIC limits
	END_IF
	cfg.aLimits_ST[i].rAlarmLow	:= MAX(cfg.aDiag[j].rAlarmLow_CPA,  cfg.aDiag[j].rAlarmLow_ESO);
	cfg.aLimits_ST[i].rAlarmHigh	:= MIN(cfg.aDiag[j].rAlarmHigh_CPA, cfg.aDiag[j].rAlarmHigh_ESO);
	cfg.aLimits_ST[i].rErrorLow	:= cfg.aDiag[j].rErrorLow;
	cfg.aLimits_ST[i].rErrorHigh	:= cfg.aDiag[j].rErrorHigh;
END_FOR
END_METHOD

END_FUNCTION_BLOCK

// POUs/Coolers/FB_CRYO_CRYOTELGT
// Cryotel GT Cooler Control
FUNCTION_BLOCK FB_CRYO_CRYOTELGT EXTENDS FB_RS_BASE
VAR_INPUT
	{attribute 'OPC.UA.DA' := '0'}
	in_bEnable:			BOOL;			// Flag to Start/Stop cooler
	{attribute 'OPC.UA.DA' := '0'}
	in_bAutoMonitor:	BOOL := TRUE;	// If true, it starts PERIODIC reads (monitoring) after INIT
	{attribute 'OPC.UA.DA' := '0'}
	in_nPeriod:			DINT := 2000;	// Interval for periodic reading [ms], default 2000 ms = 2 sec
	{attribute 'OPC.UA.DA' := '0'}
	in_sCmdSuffix:		STRING(16) := '$0D';
	{attribute 'OPC.UA.DA' := '0'}
	in_sReplySuffix:	STRING(16) := '$0D';
END_VAR
VAR_OUTPUT
END_VAR
VAR

	{attribute 'OPC.UA.DA' := '0'}
	comm:		FB_RS_COMM_CRYOTELGT;	// FB_RS_COMM_NO_SIM;		// No simulation yet
	
	// Pointers to structures inside FB_RS_COMM, e.g. ptrCommCfg.
	{attribute 'OPC.UA.DA' := '0'}
	ptrCommCfg:		POINTER TO T_RS_COMM_CFG;	(* Pointer to comm.cfg instance *)
	{attribute 'OPC.UA.DA' := '0'}
	ptrCommCtrl:	POINTER TO T_RS_COMM_CTRL;	(* Pointer to comm.ctrl instance *)
	{attribute 'OPC.UA.DA' := '0'}
	ptrCommStat:	POINTER TO T_RS_COMM_STAT;	(* Pointer to comm.stat instance *)
	
	
	{attribute 'OPC.UA.DA' := '0'}
	cfg:			T_CRYO_CRYOTELGT_CFG;	
	{attribute 'OPC.UA.DA' := '0'}
	ctrl:			T_CRYO_CRYOTELGT_CTRL;	
	{attribute 'OPC.UA.DA' := '0'}
	stat:			T_CRYO_CRYOTELGT_STAT;	

	// Pointers to arrays of INIT and READ commands
	{attribute 'OPC.UA.DA' := '0'}
	ptrInitCmds:	POINTER TO ARRAY [1..8]  OF T_CRYO_CRYOTELGT_CMD;(* Pointer to INIT commands *)
	{attribute 'OPC.UA.DA' := '0'}
	ptrReadCmds:	POINTER TO ARRAY [1..16] OF T_CRYO_CRYOTELGT_CMD;(* Pointer to READ commands *)


	(* Timers *)
	{attribute 'OPC.UA.DA' := '0'}
	fbTimer:		TON; 	// General Timeout
	timerState:		TON;	// Timer for state changes
	
	// Triggers
	triggerStart:	R_TRIG;
	triggerStop:	F_TRIG;
	

	(* Misc internal vars *)
	{attribute 'OPC.UA.DA' := '0'}
	cmdCounter:		INT := 1;	// Position in commands table
	{attribute 'OPC.UA.DA' := '0'}
	bResult:		BOOL := FALSE;
	{attribute 'OPC.UA.DA' := '0'}
	bStarted:		BOOL := FALSE;

	// TODO: Add Input signals in Fbs that EXTEND this FB.

	// Output signals
	q_bStart		AT %Q*:	BOOL;	// Start/Stop the cooler. Common to all.



END_VAR

// Hard-coded configuration
M_Configure();

(* Execute comm instance *)
M_ExecuteComm();
//comm(in_sCmdSuffix:=in_sCmdSuffix, in_sReplySuffix:=in_sReplySuffix, in_nTimeout:=3000);

// Update cooler status from digital signals.
M_UpdateStatus();

// Capture Start/Stop commands and execute the State Machine
M_StateMachine();

// Execute the base class object FB_RS_BASE
SUPER^();

METHOD ActivityInitializing
VAR_INPUT
	bExecute:	BOOL;
END_VAR
VAR_INST
	{attribute 'OPC.UA.DA' := '0'}
    nMethodState:	INT := 0;	// State Machine current state
END_VAR
VAR
	bReadOK:	BOOL;
END_VAR
SetAction('ActivityInitializing');


IF NOT bExecute THEN
	nMethodState	:= 0;	// Reset the state machine
	cmdCounter		:= 0;	// Init will start from the first init command after increment
	RETURN;
END_IF

// Handle State Machine
CASE nMethodState OF
	0:	// Set initial state and status
		stat.bInitialised	:= FALSE;
		stat.sReply			:= '';
		SetStatus(E_SM_ERROR.OK, 'BUSY');

		nMethodState := 10;				// Go to next state, i.e. INIT_COMM

	10:	// Initialize COMM port
		(* Reset the serial port *)
		ptrCommCtrl^.nCommand	:= E_RS_COMM_CMD.INIT;
		ptrCommCtrl^.bExecute	:= TRUE;

		(* Start the timer by going false/true *)
		fbTimer (IN := FALSE); (* Reset timer *)
		fbTimer (IN := TRUE, PT := T#5S); (* 5 sec timeout for reply *)

		nMethodState 	:= 15;	// On next cycle wait until the comm port is reset, i.e. idle
		
	15:	// Wait IDLE
		fbTimer (IN := TRUE);
		IF comm.stat.nStatus = E_RS_COMM_STATUS.IDLE THEN
			// Communication is IDLE 
			fbTimer (IN := FALSE);	// disable timer 
			stat.sReply		:= ptrCommStat^.sReply;	// Save the reply

			// Read from the reply.
			// Argument TRUE means that this is an INIT command.
			bReadOK	:= M_ReadFromReply(cmdCounter, TRUE);
			IF NOT bReadOK	THEN
				cmdCounter		:= 0;	// Reset command counter
				nMethodState 	:= 10;	// Wait for INIT
			ELSE
				cmdCounter		:= cmdCounter + 1;	// Increment init command index
				fbTimer (IN := FALSE);	// disable timer 
				fbTimer (IN := TRUE, PT := cfgRef.tDelay_Init); // Wait INIT delay
				bCommProblem	:= FALSE;
				nMethodState 	:= 18;	// Execute next device INIT command
			END_IF
		ELSIF comm.stat.nStatus = E_RS_COMM_STATUS.ERROR THEN
			fbTimer (IN := FALSE);
			SetStatus(E_LAKESHORE_ERROR.COMM, 'ERROR: Communication error');	
			bCommProblem	:= TRUE;
			nEvent := E_SM_EVENT.ERRINIT;
			RETURN;
		ELSIF fbTimer.Q THEN
			// Timer expired after 5 sec. This is an error.
			fbTimer (IN := FALSE);
			SetStatus(E_LAKESHORE_ERROR.TIMEOUT, 'ERROR: Communication timeout');	
			bCommProblem	:= TRUE;
			nEvent := E_SM_EVENT.ERRINIT;
			RETURN;
		END_IF

	
	
	18:	// Wait INIT Delay
		fbTimer (IN := TRUE);
		IF fbTimer.Q THEN
			// Timer expired after 5 sec. This is an error.
			fbTimer (IN := FALSE);
			nMethodState 	:= 20;	// Execute next device INIT command
			RETURN;
		END_IF

	
	
	20:	// INIT DEV
		IF ptrInitCmds^ [cmdCounter].cmd = '' THEN
			// Device INIT is done. Go to IDLE 
			stat.bInitialised 	:= TRUE;
			cmdCounter			:= 1;
			SetStatus(E_SM_ERROR.OK, 'IDLE');
			nEvent 		:= E_SM_EVENT.INITDONE;
			RETURN;
		END_IF
		
		(* Send INIT command with index cmdCounter *)
		ptrCommCtrl^.nCommand		:= E_RS_COMM_CMD.SEND;
		ptrCommCtrl^.sCmd			:= ptrInitCmds^ [cmdCounter].cmd;
		ptrCommCtrl^.nNumReplies	:= ptrInitCmds^ [cmdCounter].nReplies;
		ptrCommCtrl^.bHasReply		:= ptrInitCmds^ [cmdCounter].nReplies > 0;
		ptrCommCtrl^.bExecute		:= TRUE;
	
		(* Start the timer by going false/true *)
		fbTimer (IN := FALSE); (* Reset timer *)
		fbTimer (IN := TRUE, PT := T#5S); (* 5 sec timeout for reply *)

		// On next cycle wait until the comm port is idle
		nMethodState 	:= 15;	// On next cycle wait until the comm port is idle
	
END_CASE
END_METHOD

METHOD ActivityInitializing_new
VAR_INPUT
	bExecute:	BOOL;
END_VAR
VAR_INST
	{attribute 'OPC.UA.DA' := '0'}
    nMethodState:	INT := 0;	// State Machine current state
	{attribute 'OPC.UA.DA' := '0'}
	bCommInit:		BOOL;
END_VAR
VAR
	bReadOK:	BOOL;
END_VAR
SetAction('ActivityInitializing');


IF NOT bExecute THEN
	nMethodState	:= 0;	// Reset the state machine
	cmdCounter		:= 0;	// Init will start from the first init command after increment
	RETURN;
END_IF

// Handle State Machine
CASE nMethodState OF
	0:	// Set initial state and status
		stat.bInitialised	:= FALSE;
		stat.sReply			:= '';
		SetStatus(E_SM_ERROR.OK, 'BUSY');

		nMethodState := 10;				// Go to next state, i.e. INIT_COMM

	10:	// Initialize COMM port
		(* Reset the serial port *)
		ptrCommCtrl^.nCommand	:= E_RS_COMM_CMD.INIT;
		ptrCommCtrl^.bExecute	:= TRUE;

		(* Start the timer by going false/true *)
		fbTimer (IN := FALSE); (* Reset timer *)
		fbTimer (IN := TRUE, PT := T#5S); (* 5 sec timeout for reply *)

		bCommInit		:= TRUE;
		nMethodState 	:= 15;	// On next cycle wait until the comm port is reset, i.e. idle
		
	15:	// Wait IDLE
		fbTimer (IN := TRUE);
		IF comm.stat.nStatus = E_RS_COMM_STATUS.IDLE THEN
			// If we have just executed the COMM Reset/INIT command,
			// Go to first INIT command.
			IF bCommInit THEN
				bCommInit		:= FALSE;
				cmdCounter		:= 1;	// Start from first INIT command
				fbTimer (IN := FALSE);	// disable timer 
				fbTimer (IN := TRUE, PT := cfgRef.tDelay_Init); // Wait INIT delay
				bCommProblem	:= FALSE;
				nMethodState 	:= 18;	// Execute next device INIT command
				RETURN;
			END_IF
			// Communication is IDLE 
			fbTimer (IN := FALSE);	// disable timer 
			stat.sReply		:= ptrCommStat^.sReply;	// Save the reply

			// Read from the reply.
			// Argument TRUE means that this is an INIT command.
			bReadOK	:= M_ReadFromReply(cmdCounter, TRUE);
			IF NOT bReadOK	THEN
				cmdCounter		:= 0;	// Reset command counter
				nMethodState 	:= 10;	// Wait for INIT
			ELSE
				cmdCounter		:= cmdCounter + 1;	// Increment init command index
				fbTimer (IN := FALSE);	// disable timer 
				fbTimer (IN := TRUE, PT := cfgRef.tDelay_Init); // Wait INIT delay
				bCommProblem	:= FALSE;
				nMethodState 	:= 18;	// Execute next device INIT command
			END_IF
		ELSIF comm.stat.nStatus = E_RS_COMM_STATUS.ERROR THEN
			fbTimer (IN := FALSE);
			SetStatus(E_LAKESHORE_ERROR.COMM, 'ERROR: Communication error');	
			bCommProblem	:= TRUE;
			nEvent := E_SM_EVENT.ERRINIT;
			RETURN;
		ELSIF fbTimer.Q THEN
			// Timer expired after 5 sec. This is an error.
			fbTimer (IN := FALSE);
			SetStatus(E_LAKESHORE_ERROR.TIMEOUT, 'ERROR: Communication timeout');	
			bCommProblem	:= TRUE;
			nEvent := E_SM_EVENT.ERRINIT;
			RETURN;
		END_IF

	
	
	16:	// Delay and then goto Wait for IDLE
		fbTimer (IN := TRUE);

		IF fbTimer.Q THEN
			fbTimer (IN := FALSE); // Reset timer
			fbTimer (IN := TRUE, PT := T#5S);	// 5sec timeout for reply.	
			nMethodState 	:= 15;	// Goto Wait for IDLE
			RETURN;
		END_IF
	
	18:	// Delay and then goto execute next command
		fbTimer (IN := TRUE);
		IF fbTimer.Q THEN
			// Timer expired after 5 sec. This is an error.
			fbTimer (IN := FALSE);
			nMethodState 	:= 20;	// Goto next INIT command
			RETURN;
		END_IF

	
	
	20:	// INIT DEV
		IF ptrInitCmds^ [cmdCounter].cmd = '' THEN
			// Device INIT is done. Go to IDLE 
			stat.bInitialised 	:= TRUE;
			cmdCounter			:= 1;
			SetStatus(E_SM_ERROR.OK, 'IDLE');
			nEvent 		:= E_SM_EVENT.INITDONE;
			RETURN;
		END_IF
		
		(* Send INIT command with index cmdCounter *)
		ptrCommCtrl^.nCommand		:= E_RS_COMM_CMD.SEND;
		ptrCommCtrl^.sCmd			:= ptrInitCmds^ [cmdCounter].cmd;
		ptrCommCtrl^.nNumReplies	:= ptrInitCmds^ [cmdCounter].nReplies;
		ptrCommCtrl^.bHasReply		:= ptrInitCmds^ [cmdCounter].nReplies > 0;
		ptrCommCtrl^.bExecute		:= TRUE;
	
		// In case this is a command without a reply,
		// we apply 200ms delay between commmands.
		IF NOT ptrCommCtrl^.bHasReply THEN
			// There is no reply, i.e. this is a 'SET' command.
			// Start the timer by going false/true.
			// Apply 200ms delay between SET commands.
			fbTimer (IN := FALSE); // Reset timer
			fbTimer (IN := TRUE, PT := T#200MS); 
			cmdCounter		:= cmdCounter + 1;	// Go to next command.
			nMethodState	:= 18;				// Goto WAIT for delay.
			RETURN;
		ELSE			
			// There is a reply.
			// Apply a delay of 20ms before checking the status. 
			// Start the timer by going false/true
			fbTimer (IN := FALSE); // Reset timer
			fbTimer (IN := TRUE, PT := T#5MS);	
			stat.sErrorText	:= 'BUSY';
			nMethodState := 16;	// Goto WAIT for Reading to complete,
		END_IF
		
END_CASE
END_METHOD

METHOD ActivityMonitoring
VAR_INPUT
	bExecute:	BOOL;
END_VAR
VAR_INST
	{attribute 'OPC.UA.DA' := '0'}
    nMethodState:	INT := 0;	// State Machine current state
	{attribute 'OPC.UA.DA' := '0'}
	nRetries:		INT := 0;	// Number of retries in case of communication problems
END_VAR

VAR
	offset: INT;
	bReadOK:	BOOL;
END_VAR
IF NOT cfgRef.bAutoMonitor AND stat.nSubstate = E_RS_BASE_SUBSTATE.NOTOP_READY THEN
	SetAction('No Monitoring'); 
	SetStatus(E_SM_ERROR.OK, 'IDLE');
	nMethodState	:= 0;	// Reset the state machine
	cmdCounter		:= 1;	// Reading will start from the first command in the array
	RETURN;
END_IF

IF NOT bExecute THEN
	SetAction('ActivityMonitoring'); 
	SetStatus(E_SM_ERROR.OK, 'BUSY');
	nMethodState	:= 0;	// Reset the state machine
	cmdCounter		:= 1;	// Reading will start from the first command in the array
	RETURN;
END_IF

// Handle State Machine
CASE nMethodState OF
	0:	// Execute a command from the command array
		IF ptrReadCmds^ [cmdCounter].cmd = '' OR cmdCounter > 16 THEN

			// All commands have been executed. 
			// Wait tDelay_Periodic before re-starting the READ.
			cmdCounter	:= 1;
			SetStatus(E_SM_ERROR.OK, 'IDLE');
			
			(* Start the timer by going false/true *)
			fbTimer (IN := FALSE); (* Reset timer *)
			fbTimer (IN := TRUE, PT := cfgRef.tDelay_Periodic);
			nMethodState := 10;				// Goto Wait for tDelay_Periodic
			RETURN;
			
		END_IF
		
		(* Send command with index cmdCounter *)
		ptrCommCtrl^.nCommand		:= E_RS_COMM_CMD.SEND;
		ptrCommCtrl^.sCmd			:= ptrReadCmds^ [cmdCounter].cmd;
		ptrCommCtrl^.nNumReplies	:= ptrReadCmds^ [cmdCounter].nReplies;
		ptrCommCtrl^.bHasReply		:= ptrReadCmds^ [cmdCounter].nReplies > 0;
		ptrCommCtrl^.bExecute		:= TRUE;
		
		// In case we are executing 'SET' commands, there are no replies.
		// However, we need a delay of at least 50ms between commands.
		// We will apply 150ms.
		IF NOT ptrCommCtrl^.bHasReply THEN
			// There is no reply, i.e. this is a 'SET' command.
			// Start the timer by going false/true.
			// Apply 200ms delay between SET commands.
			fbTimer (IN := FALSE); // Reset timer
			fbTimer (IN := TRUE, PT := T#200MS); 
			cmdCounter		:= cmdCounter + 1;	// Go to next command.
			nMethodState	:= 10;				// Goto WAIT for Reading to complete,
			RETURN;
		ELSE			
			// There is a reply, i.e. this is a 'READ' command.
			// Apply a delay of 10ms before checking the status. 
			// Start the timer by going false/true
			fbTimer (IN := FALSE); // Reset timer
			fbTimer (IN := TRUE, PT := T#10MS);	
			stat.sErrorText	:= 'BUSY';
			nMethodState := 15;	// Goto WAIT for Reading to complete,
		END_IF
		

	10:	// Wait until the delay timeout expires
		fbTimer (IN := TRUE);

		(* If Timer has expired, go to the next state. *)
		IF fbTimer.Q THEN
			fbTimer (IN := FALSE);
			nMethodState 	:= 0;	// Goto Wait for tDelay_Periodic
			RETURN;
		END_IF
	
	15:	// Wait until the delay timeout expires
		fbTimer (IN := TRUE);

		(* If Timer has expired, go to the next state. *)
		IF fbTimer.Q THEN
			fbTimer (IN := FALSE);
			fbTimer (IN := TRUE, PT := T#5S);	// 5 sec timeout for reply
			stat.sErrorText	:= 'BUSY';
			nMethodState 	:= 20;	// Goto Wait for IDLE/Reply
			RETURN;
		END_IF
	



	20:	// Wait for the reading to complete, i.e. IDLE
		fbTimer (IN := TRUE);
		IF comm.stat.nStatus = E_RS_COMM_STATUS.IDLE THEN
			// Communication is IDLE 
			fbTimer (IN := FALSE);	// disable timer 
			stat.sReply		:= ptrCommStat^.sReply;	// Save the reply
			
			// Copy readings to status variable(s)
			
			// Read from the reply.
			// Argument FALSE means that this is NOT an INIT command.
			bReadOK	:= M_ReadFromReply(cmdCounter, FALSE);
			IF NOT bReadOK	THEN
				// Reply was not OK. Maybe out of sync.
				// Re-INIT the communication, i.e. clear the buffer.
				ptrCommCtrl^.nCommand	:= E_RS_COMM_CMD.INIT;
				ptrCommCtrl^.bExecute	:= TRUE;
		
				(* Start the timer by going false/true *)
				fbTimer (IN := FALSE); (* Reset timer *)
				fbTimer (IN := TRUE, PT := T#5S); (* 5 sec timeout for reply *)
		
				SetStatus(E_LAKESHORE_ERROR.COMM, 'ERROR: Communication error');	
				bCommProblem	:= TRUE;

				nMethodState 	:= 10;	// On next cycle wait until the comm port is reset, i.e. idle
				RETURN;
			ELSE
				// All OK. Go to next command.
				bCommProblem	:= FALSE;
				nRetries		:= 0;	// Reset number of retries
		
				cmdCounter		:= cmdCounter + 1;	// Go to next command.
				
				// Apply a 150 ms delay between commands
				fbTimer (IN := FALSE);	// Reset timer
				fbTimer (IN := TRUE, PT := cfg.tDelay_Read); 
				nMethodState := 10;		// Apply delay
				nEvent := E_SM_EVENT.COMMOK;
				RETURN;
			END_IF
		ELSIF comm.stat.nStatus = E_RS_COMM_STATUS.ERROR OR fbTimer.Q THEN
			// No Reply.
			// Re-INIT the communication, i.e. clear the buffer.
			ptrCommCtrl^.nCommand	:= E_RS_COMM_CMD.INIT;
			ptrCommCtrl^.bExecute	:= TRUE;
	
			(* Start the timer by going false/true *)
			fbTimer (IN := FALSE); (* Reset timer *)
			fbTimer (IN := TRUE, PT := T#5S); (* 5 sec timeout for reply *)
	
			SetStatus(E_LAKESHORE_ERROR.COMM, 'ERROR: Communication error');	
			bCommProblem	:= TRUE;

			nRetries		:= nRetries + 1;		// Increment number of retries
			stat.nRetries	:= stat.nRetries + 1;	// Increment total number of retries

			nMethodState 	:= 10;	// On next cycle wait until the comm port is reset, i.e. idle
			RETURN;
		END_IF

	
END_CASE
END_METHOD

METHOD M_AddCtrlCommands : BOOL
VAR_INPUT
//	in_sCmd:	STRING;
END_VAR
VAR
	i:	INT;
    fbFormat:	FB_FormatString;
	nVal:		UDINT;
	lrVal:		LREAL;
	sPowerCmd:	STRING;
END_VAR
// Find index of first two empty commands.
// The result must be greater than zero, if everuthing is OK.
i	:= M_FindReadCommand('');

// Add relevant control commands to the end of the list
// of Read/status comands.
IF i > 0	THEN
	IF ctrl.nDevCmd	= E_CRYO_CRYOTELGT_CMD.ON	THEN
		// Cooler is always started with 240W output.
		// Write the output power and then the ON command.
		ctrl.lrPower	:= 240.0;
		cfg.cmdList_Read[i].cmd			:= 'PWOUT=240';
		cfg.cmdList_Read[i+1].cmd		:= 'COOLER=POWER';
		// Each command has a single reply.
		cfg.cmdList_Read[i].nReplies	:= 2;
		cfg.cmdList_Read[i+1].nReplies	:= 2;
	ELSIF ctrl.nDevCmd	= E_CRYO_CRYOTELGT_CMD.OFF	THEN
		// Write the power OFF command.
		cfg.cmdList_Read[i].cmd			:= 'COOLER=OFF';
		cfg.cmdList_Read[i+1].cmd		:= '';
		// Each command has a single reply.
		cfg.cmdList_Read[i].nReplies	:= 2;
		cfg.cmdList_Read[i+1].nReplies	:= 0;
	ELSIF ctrl.nDevCmd	= E_CRYO_CRYOTELGT_CMD.SET_POWER	THEN
		// Updating only the power value.
		ctrl.bPower	:= TRUE;
		// Write the output power command.
		lrVal	:= ctrl.lrPower;
		fbFormat(	sFormat := 'PWOUT=%.2f', 
					arg1 := F_LREAL(lrVal), 
					sOut => sPowerCmd);
		cfg.cmdList_Read[i].cmd			:= sPowerCmd;
		cfg.cmdList_Read[i+1].cmd		:= '';
		// Each command has a single reply.
		cfg.cmdList_Read[i].nReplies	:= 2;
		cfg.cmdList_Read[i+1].nReplies	:= 0;
	END_IF
	
	M_AddCtrlCommands	:= TRUE;
ELSE
	M_AddCtrlCommands	:= FALSE;
END_IF
END_METHOD

METHOD M_ClearCtrlCommands
VAR_INPUT
END_VAR
VAR
	i:	INT;
END_VAR
// Search for commands starting with  'COOLER=' and 'PWOUT='.
// If found, clear them.
FOR i := 1 TO 16 DO
	IF FIND(cfg.cmdList_Read[i].cmd, 'PWOUT=') > 0	THEN
		cfg.cmdList_Read[i].cmd	:= '';
	ELSIF FIND(cfg.cmdList_Read[i].cmd, 'COOLER=') > 0	THEN
		cfg.cmdList_Read[i].cmd	:= '';
	END_IF
END_FOR

ctrl.nDevCmd	:= E_CRYO_CRYOTELGT_CMD.NONE;
ctrl.bPower		:= FALSE;
END_METHOD

METHOD M_Configure
VAR_INPUT
END_VAR
VAR
		i:	INT;
END_VAR
IF NOT bStarted	THEN
	//
	// START: Mandatory  !!!
	//
	// Set references from FB_RS_BASE
	cfgRef	REF=cfg;
	ctrlRef	REF=ctrl;
	statRef	REF=stat;

	// Ensure that the references are correctly set
	IF	NOT __ISVALIDREF(cfgRef)	OR  
		NOT __ISVALIDREF(ctrlRef)	OR  
		NOT __ISVALIDREF(statRef)		THEN
		stat.sErrorText	:= 'References not configured';
		RETURN;
	END_IF
	
	// Copy input parameters to configuration
	cfg.bAutoMonitor	:= in_bAutoMonitor;
	cfg.tDelay_Periodic	:= DINT_TO_TIME(in_nPeriod);
	cfg.tDelay_Ctrl		:= T#200MS;
	
	
	// Set pointers to arrays of commands
	ptrInitCmds	:= ADR(cfg.cmdList_Init);(* Pointer to INIT commands *)
	ptrReadCmds	:= ADR(cfg.cmdList_Read);(* Pointer to READ commands *)
	
	// TODO in FB that extends the functionality
	// Set pointers to comm, i.e.
	ptrCommCfg	:= ADR(comm.cfg);	(* Pointer to comm.cfg instance *)
	ptrCommCtrl	:= ADR(comm.ctrl);	(* Pointer to comm.ctrl instance *)
	ptrCommStat	:= ADR(comm.stat);	(* Pointer to comm.stat instance *)
	
	// Set comm suffixes for commands and replies
	ptrCommCfg^.sCmdSuffix		:= in_sCmdSuffix;
	ptrCommCfg^.sReplySuffix	:= in_sReplySuffix;

	stat.bConfigured	:= TRUE;
	bStarted			:= TRUE;
	//
	// END: Mandatory for ALL cooler !!!
	//


	
END_IF
END_METHOD

METHOD M_ExecuteComm
VAR_INPUT
END_VAR
comm(	in_bSimulation	:= in_bSimulation, 
		in_sCmdSuffix	:= in_sCmdSuffix, 
		in_sReplySuffix	:= in_sReplySuffix, 
		in_nTimeout		:= 3000);
END_METHOD

// Return the index of the command in cfg.cmdList_Read[].
// Returns zero if not found.
METHOD M_FindReadCommand : INT
VAR_INPUT
	in_sCmd:	STRING;
END_VAR
VAR
	i:	INT;
END_VAR
// We need two empty commands: 'COOLER=<>' and 'PWOUT=<VAL>'.
// Thats's why the highest index is 15 rather than 16.
FOR i := 1 TO 15 DO
	IF cfg.cmdList_Read[i].cmd = in_sCmd	THEN
		M_FindReadCommand	:= i;
		RETURN;
	END_IF
END_FOR

M_FindReadCommand	:= 0;
END_METHOD

METHOD M_GetCouplerState : BOOL
VAR_INPUT
END_VAR
IF comm.i_nCouplerState = 8  OR  comm.in_bSimulation  THEN
	M_GetCouplerState	:= TRUE;	
ELSE
	M_GetCouplerState	:= FALSE;	
END_IF
END_METHOD

METHOD M_ReadFromReply : BOOL
// Method to check correctness of the reply and assign the result to a status variable.
VAR_INPUT
	idx:		INT;			// Command index in the array.
	bInitCmd:	BOOL := FALSE;	// If TRUE, this is an INIT command, otherwise it is Read/status
END_VAR
VAR
	pos:	INT;
	length:	INT;
	cmd:	STRING;
	subStr:	STRING;
END_VAR
// During INIT it might happen that the command index is 0.
// These cases should be discarded.
IF idx <= 0	THEN
	M_ReadFromReply	:= TRUE;
	RETURN;
END_IF

// Get the command
IF bInitCmd	THEN
	cmd		:= cfg.cmdList_Init[idx].cmd;
ELSE
	cmd		:= cfg.cmdList_Read[idx].cmd;
END_IF

// The sent command has to be included in the first line of the reply.
// If not, we are out of sync and have to reinitialise.
IF FIND(stat.sReply, cmd) = 0	THEN
	bCommProblem	:= TRUE;
	stat.nState		:= E_RS_BASE_STATE.NOTOP;
	stat.nSubstate	:= E_RS_BASE_SUBSTATE.NOTOP_NOTREADY;
	RETURN;
END_IF

// Extract the value from the reply.
// Example: 
//    Command: VERSION
//    Reply:   VERSION$R$Nv1.4.1$R
//    Value:   v1.4.1
//
// Take the string after the '$R$N' and remove the '$R' at the end.
// Remove the <CR> suffix from the reply.

pos	:= FIND(stat.sReply,'$R$N');
IF pos = 0	THEN
	// The string is not found. 
	M_ReadFromReply	:= FALSE;
	RETURN;
END_IF

length	:= LEN(stat.sReply) - pos -2;
subStr	:= MID(stat.sReply, length, pos+2);


IF cmd = 'VERSION'	THEN
	stat.sVersion	:= subStr;
ELSIF cmd = 'MODE'	THEN
	stat.sMode		:= subStr;
ELSIF cmd = 'SENSOR'	THEN
	stat.sSensor	:= subStr;
ELSIF FIND(cmd, 'PWOUT=') = 1	THEN
	// Get the commanded power from the command.
	// Get the value after the 'PWOUT=' substring.
	stat.lrPowerCommanded	:= STRING_TO_LREAL(subStr);
	// If we are updating only the power value,
	// this is then the last control command.
	IF ctrl.bPower	THEN
		// Clear the control commands from the list.
		M_ClearCtrlCommands();
		ctrl.bPower	:= FALSE;
		// Power output command is not active any more.
		stat.bPowerCmdActive	:= FALSE;
	END_IF
ELSIF FIND(cmd, 'COOLER=') = 1	THEN
	// Get the control mode 'POWER' or 'OFF'.
	stat.sCtrlMode	:= subStr;
	// This is the last control command when switching cool on/off.
	// Clear the control commands from the list.
	M_ClearCtrlCommands();
	// Power output command is not active any more.
	stat.bPowerCmdActive	:= FALSE;
ELSIF cmd = 'ERROR'	THEN
	IF FIND(subStr, '00000001') = 1	THEN
		stat.sCtrlError	:= 'High Reject Temperature';
	ELSIF FIND(subStr, '00000010') = 1	THEN
		stat.sCtrlError	:= 'Low Reject Temperature';
	ELSIF FIND(subStr, '10000000') = 1	THEN
		stat.sCtrlError	:= 'Over Current Error';
	ELSIF FIND(subStr, '11111111') = 1	THEN
		stat.sCtrlError	:= 'Invalid Configuration';
	ELSE
		stat.sCtrlError	:= 'OK';
	END_IF
ELSIF cmd = 'COOLER'	THEN
	stat.sCtrlMode	:= subStr;
ELSIF cmd = 'P'	THEN
	stat.lrPowerMeasured	:= STRING_TO_LREAL(subStr);
ELSIF cmd = 'PWOUT'	THEN
	stat.lrPowerCommanded	:= STRING_TO_LREAL(subStr);
ELSIF cmd = 'TC'	THEN
	stat.lrTempColdHead		:= STRING_TO_LREAL(subStr);
ELSIF cmd = 'TEMP RJ'	THEN
	stat.lrTempReject		:= STRING_TO_LREAL(subStr);
ELSIF cmd = 'TTARGET'	THEN
	stat.lrTempTarget		:= STRING_TO_LREAL(subStr);
END_IF


M_ReadFromReply	:= TRUE;	// OK
END_METHOD

METHOD M_StateMachine
VAR_INPUT
END_VAR
//////////////////////
// Cooler State Machine
//////////////////////
CASE stat.nDevState OF
	E_CRYO_CRYOTELGT_STATE.OFF:
		// Capture START command when in_bEnable goes TRUE.
		triggerStart(CLK:=in_bEnable);
		IF triggerStart.Q	THEN
			// in_bEnable is TRUE, start the cooler.
			ctrl.bStart		:= TRUE;	// For digital control. Not used currently.
			ctrl.nDevCmd	:= E_CRYO_CRYOTELGT_CMD.ON;
			M_AddCtrlCommands();	// Add ON related commands
			stat.nDevState	:= 	E_CRYO_CRYOTELGT_STATE.STARTING;
			stat.sDevState	:= 'Starting...';
			// Restart the timer
			timerState(IN:=FALSE);
			timerState(IN:=TRUE,PT:=UDINT_TO_TIME(cfg.nTimeoutState));
		END_IF
	E_CRYO_CRYOTELGT_STATE.STARTING:
		timerState();	// Timeout for the state transition.
		triggerStop(CLK:= in_bEnable);	// Check if the cooler should be switched OFF.
		IF timerState.Q THEN
			// Timeout, stop the cooler.
			ctrl.bStart		:= FALSE;
			timerState(IN:=FALSE);
			M_ClearCtrlCommands();	// Clear ON related commands
			stat.nDevState	:= 	E_CRYO_CRYOTELGT_STATE.ERROR;
			stat.sDevState	:= 'ERROR - Timeout on START';
		ELSIF stat.sCtrlMode = 'POWER' THEN
			// State is 'POWER'.
			// That means that the cooler is ON in power mode.
			timerState(IN:=FALSE);
			M_ClearCtrlCommands();	// Clear ON related commands
			stat.nDevState	:= 	E_CRYO_CRYOTELGT_STATE.ON;
			stat.sDevState	:= 'ON';
		ELSIF triggerStop.Q THEN
			// in_bEnable is FALSE, stop the cooler.
			ctrl.bStart		:= FALSE;
			ctrl.nDevCmd	:= E_CRYO_CRYOTELGT_CMD.OFF;
			ctrl.lrPower	:= 240.0;
			M_ClearCtrlCommands();	// Clear ON related commands
			M_AddCtrlCommands();	// Add OFF related commands
			// Restart the timer
			timerState(IN:=FALSE);
			timerState(IN:=TRUE,PT:=UDINT_TO_TIME(cfg.nTimeoutState));
			stat.nDevState	:= 	E_CRYO_CRYOTELGT_STATE.STOPPING;
			stat.sDevState	:= 'Stopping...';
		END_IF
	E_CRYO_CRYOTELGT_STATE.ON:
		triggerStop(CLK:= in_bEnable);
		IF triggerStop.Q THEN
			// in_bEnable is FALSE, stop the cooler.
			// Restart the timer for state transition.
			ctrl.bStart		:= FALSE;
			ctrl.nDevCmd	:= E_CRYO_CRYOTELGT_CMD.OFF;
			M_AddCtrlCommands();	// Add OFF related commands
			timerState(IN:=FALSE);
			timerState(IN:=TRUE,PT:=UDINT_TO_TIME(cfg.nTimeoutState));
			stat.nDevState	:= 	E_CRYO_CRYOTELGT_STATE.STOPPING;
			stat.sDevState	:= 'Stopping...';
		ELSIF stat.sCtrlMode <> 'POWER' THEN
			// 'POWER' is the only operational mode.
			// If it is something else, stop the cooler.
			ctrl.bStart		:= FALSE;
			ctrl.nDevCmd	:= E_CRYO_CRYOTELGT_CMD.OFF;
			M_AddCtrlCommands();	// Add OFF related commands
			stat.nDevState	:= 	E_CRYO_CRYOTELGT_STATE.ERROR;
			stat.sDevState	:= 'ERROR - Unexpected OFF';
		ELSIF stat.lrTempColdHead < 100.0  AND ctrl.lrPower < 250.0	THEN
			// Switch the power to 250W if the cold head temperature is below 100K.
			IF NOT stat.bPowerCmdActive	THEN
				stat.bPowerCmdActive	:= TRUE;
				ctrl.lrPower			:= 250.0;
				ctrl.nDevCmd			:= E_CRYO_CRYOTELGT_CMD.SET_POWER;
				M_AddCtrlCommands();	// Add OFF related commands
			END_IF
		ELSIF stat.lrTempColdHead > 101.0  AND ctrl.lrPower > 240.0	THEN
			// Switch the power to 240W if the cold head temperature is above 101K.
			IF NOT stat.bPowerCmdActive	THEN
				stat.bPowerCmdActive	:= TRUE;
				ctrl.lrPower			:= 240.0;
				ctrl.nDevCmd			:= E_CRYO_CRYOTELGT_CMD.SET_POWER;
				M_AddCtrlCommands();	// Add OFF related commands
			END_IF
		END_IF
	E_CRYO_CRYOTELGT_STATE.STOPPING:
		timerState();
		// Capture START command
		triggerStart(CLK:=in_bEnable);
		IF timerState.Q THEN
			timerState(IN:=FALSE);
			M_ClearCtrlCommands();	// Clear OFF related commands
			stat.nDevState	:= 	E_CRYO_CRYOTELGT_STATE.ERROR;
			stat.sDevState	:= 'ERROR - Timeout on STOP';
		ELSIF stat.sCtrlMode = 'OFF' THEN
			timerState(IN:=FALSE);
			M_ClearCtrlCommands();	// Clear OFF related commands
			stat.nDevState	:= 	E_CRYO_CRYOTELGT_STATE.OFF;
			stat.sDevState	:= 'OFF';
		ELSIF triggerStart.Q THEN
			// in_bEnable is TRUE, start the cooler.
			ctrl.bStart		:= TRUE;
			M_ClearCtrlCommands();	// Clear OFF related commands
			ctrl.nDevCmd	:= E_CRYO_CRYOTELGT_CMD.ON;
			M_AddCtrlCommands();	// Add ON related commands
			stat.nDevState	:= 	E_CRYO_CRYOTELGT_STATE.STARTING;
			stat.sDevState	:= 'Starting...';
			// Restart the timer
			timerState(IN:=FALSE);
			timerState(IN:=TRUE,PT:=UDINT_TO_TIME(cfg.nTimeoutState));
		END_IF
	E_CRYO_CRYOTELGT_STATE.ERROR:
		// To recover from error, STOP command has to be issued
		// in order to reset triggerStop.
		// Capture STOP command
		triggerStop(CLK:=in_bEnable);
		IF triggerStop.Q THEN
			// in_bEnable is FALSE, stop the cooler.
			ctrl.nDevCmd	:= E_CRYO_CRYOTELGT_CMD.OFF;
			M_AddCtrlCommands();	// Add ON related commands
			stat.nDevState	:= 	E_CRYO_CRYOTELGT_STATE.STOPPING;
			stat.sDevState	:= 'OFF';
			RETURN;
		END_IF
		
		// Capture START command.
		triggerStart(CLK:=in_bEnable);
		IF triggerStart.Q THEN
			// in_bEnable is TRUE, start the cooler.
			ctrl.bStart		:= TRUE;
			ctrl.nDevCmd	:= E_CRYO_CRYOTELGT_CMD.ON;
			M_AddCtrlCommands();	// Add ON related commands
			stat.nDevState	:= 	E_CRYO_CRYOTELGT_STATE.STARTING;
			stat.sDevState	:= 'Starting...';
			// Restart the timer
			timerState(IN:=FALSE);
			timerState(IN:=TRUE,PT:=UDINT_TO_TIME(cfg.nTimeoutState));
		END_IF
END_CASE


// Update outputs
q_bStart	:= ctrl.bStart;
END_METHOD

METHOD M_UpdateStatus
VAR_INPUT
END_VAR
// TODO: For each cooler FB that extends FB_CRYO_PUMP_BASE update inputs in M_UpdateStatus(), e.g.

(*
// Update inputs
stat.bReady		:= i_bReady;
stat.bSpeed100	:= i_bSpeed100;
stat.bWarning	:= i_bWarning;
stat.bAlarm		:= i_bAlarm;

CASE stat.nCtrlMode	OF
	0:	stat.sCtrlMode	:= 'HHR (Hand-Held Remote)';
	1:	stat.sCtrlMode	:= 'REMOTE';
	2:	stat.sCtrlMode	:= 'SERIAL LINK';
	3:	stat.sCtrlMode	:= 'FIELDBUS';
ELSE
	stat.sCtrlMode	:= 'UNKNOWN';
END_CASE

*)
END_METHOD

METHOD ProcessEvents
VAR_INPUT
END_VAR

(* 
	Before processing the event, execute the Do-Activity tasks. 
	Note that, in case of orthogonal regions, more than one Do-Activity 
	could run in the same PLC cycle.
	Note: Most of these activities have timeouts since they take time.
*)

IF	statRef.nSubstate = E_RS_BASE_SUBSTATE.OP_MONITORING 		OR 
	statRef.nSubstate = E_RS_BASE_SUBSTATE.NOTOP_READY			OR
	(statRef.nSubstate = E_RS_BASE_SUBSTATE.NOTOP_ERROR 	AND 
	 nLastGoodSubstate = E_RS_BASE_SUBSTATE.NOTOP_READY) 		OR 
	(statRef.nSubstate = E_RS_BASE_SUBSTATE.OP_ERROR 		AND 
	 nLastGoodSubstate = E_RS_BASE_SUBSTATE.OP_MONITORING)			THEN
	ActivityMonitoring(TRUE);
ELSIF statRef.nSubstate = E_RS_BASE_SUBSTATE.OP_MONITORING_USER THEN
	ActivityMonitoringUser(TRUE);
ELSIF statRef.nSubstate = E_RS_BASE_SUBSTATE.NOTOP_INITIALIZING THEN
	ActivityInitializing(TRUE);
END_IF

// Set last known good substate. Used for recovery from comm problems.
M_SetLastGoodSubstate();

(* 
	Evaluate state machine transitions.
*)

CASE statRef.nState OF

//***********************************
// NOTOP
//***********************************
E_RS_BASE_STATE.NOTOP:

	(* Transitions from NOTOP substates *)
	CASE statRef.nSubstate OF
	
	E_RS_BASE_SUBSTATE.NOTOP_NOTREADY:		
		IF 	nEvent = E_SM_EVENT.INIT OR cfgRef.bAutoMonitor  THEN
			nEvent := E_SM_EVENT.INIT;
			ActionInitExecute();
			SetState(E_RS_BASE_STATE.NOTOP, E_RS_BASE_SUBSTATE.NOTOP_INITIALIZING);
			SetStatus(E_SM_ERROR.OK, 'OK');
			RETURN;
		END_IF
		
	E_RS_BASE_SUBSTATE.NOTOP_INITIALIZING:			
		IF nEvent = E_SM_EVENT.INITDONE THEN
			nReadType := E_RS_BASE_READ_TYPE.PERIODIC;
			ActivityMonitoring(FALSE);	// Reset Monitoring method
			IF cfgRef.bAutoMonitor THEN
				nEvent := E_SM_EVENT.ENABLE;
				statRef.bAutoStarted	:= TRUE;
				SetState(E_RS_BASE_STATE.OP, E_RS_BASE_SUBSTATE.OP_MONITORING);
			ELSE
				SetState(E_RS_BASE_STATE.NOTOP, E_RS_BASE_SUBSTATE.NOTOP_READY);
			END_IF
			RETURN;
		ELSIF nEvent = E_SM_EVENT.ERRINIT THEN
			// INIT failed. Keep re-trying.
			SetState(E_RS_BASE_STATE.NOTOP, E_RS_BASE_SUBSTATE.NOTOP_NOTREADY);
			RETURN;
		END_IF
		
	E_RS_BASE_SUBSTATE.NOTOP_READY:			
		IF nEvent = E_SM_EVENT.ENABLE THEN
			IF cfgRef.bAutoMonitor THEN
				// Monitoring is already in progress.
				// It has to complete the read cycle in a clean way.
				nNextState		:= E_RS_BASE_STATE.OP;					// Next state after STOP	
				nNextSubstate	:= E_RS_BASE_SUBSTATE.OP_MONITORING;	// Next substate after STOP	
				nNextDescription:= 'BUSY';
				nReadType		:= E_RS_BASE_READ_TYPE.PERIODIC;
				RETURN;
			ELSE
				SetState(E_RS_BASE_STATE.OP, E_RS_BASE_SUBSTATE.OP_MONITORING);
				// This call MUST be after SetState()
				ActivityMonitoring(FALSE);	// Reset Monitoring method
			END_IF
		END_IF

	E_RS_BASE_SUBSTATE.NOTOP_ERROR:			
		IF nEvent = E_SM_EVENT.HWOK THEN
			SetState(E_RS_BASE_STATE.NOTOP, E_RS_BASE_SUBSTATE.NOTOP_NOTREADY);
			RETURN;
		ELSIF nEvent = E_SM_EVENT.COMMOK THEN
			SetState(E_RS_BASE_STATE.NOTOP, nLastGoodSubstate);
			RETURN;			
		END_IF
		
	END_CASE

	(* Transitions from NOTOP state *)
	IF	nEvent = E_SM_EVENT.ERRHW OR
		nEvent = E_SM_EVENT.ERRCOMM	THEN
		ActionUnexpExecute();
		SetState(E_RS_BASE_STATE.NOTOP, E_RS_BASE_SUBSTATE.NOTOP_ERROR);
		RETURN;
	END_IF
	
//***********************************
// OPERATIONAL
//***********************************
E_RS_BASE_STATE.OP:

	(* Transitions from OP subastates *)
	CASE statRef.nSubstate OF
	E_RS_BASE_SUBSTATE.OP_ERROR:			
		IF 	cfgRef.bAutoMonitor  THEN
			nEvent := E_SM_EVENT.INIT;
			ActionInitExecute();
			SetState(E_RS_BASE_STATE.NOTOP, E_RS_BASE_SUBSTATE.NOTOP_INITIALIZING);
			SetStatus(E_SM_ERROR.OK, 'Recovering from error...');
			RETURN;
		END_IF
		IF nEvent = E_SM_EVENT.HWOK THEN
			SetStatus(E_SM_ERROR.OK, 'OK');
			SetState(E_RS_BASE_STATE.OP, E_RS_BASE_SUBSTATE.OP_IDLE);
			RETURN;			
		ELSIF nEvent = E_SM_EVENT.DISABLE THEN
			ActionDisableExecute();
			SetState(E_RS_BASE_STATE.NOTOP, E_RS_BASE_SUBSTATE.NOTOP_ERROR);
			RETURN;			
		ELSIF nEvent = E_SM_EVENT.COMMOK THEN
			SetState(E_RS_BASE_STATE.OP, nLastGoodSubstate);
			RETURN;			
		END_IF

	E_RS_BASE_SUBSTATE.OP_MONITORING:
		IF nEvent = E_SM_EVENT.DISABLE THEN
			ActionDisableExecute();
			RETURN;			
		ELSIF nEvent = E_SM_EVENT.STOPMON THEN
			ActionStopExecute();
			RETURN;			
		ELSIF nEvent = E_SM_EVENT.READDONE THEN
			SetState(E_RS_BASE_STATE.OP, E_RS_BASE_SUBSTATE.OP_IDLE);
			RETURN;			
		ELSIF nEvent = E_SM_EVENT.ERRCOMM THEN
			SetState(E_RS_BASE_STATE.OP, E_RS_BASE_SUBSTATE.OP_ERROR);
			RETURN;			
		END_IF
		
	E_RS_BASE_SUBSTATE.OP_MONITORING_USER:			
		IF nEvent = E_SM_EVENT.DISABLE THEN
			ActionDisableExecute();
			RETURN;			
		ELSIF nEvent = E_SM_EVENT.STOPMON THEN
			ActionStopExecute();
			RETURN;			
		ELSIF nEvent = E_SM_EVENT.READDONE THEN
			SetState(E_RS_BASE_STATE.OP, E_RS_BASE_SUBSTATE.OP_IDLE);
			RETURN;			
		END_IF
		
	E_RS_BASE_SUBSTATE.OP_IDLE:			
		IF nEvent = E_SM_EVENT.DISABLE THEN
			ActionDisableExecute();
			RETURN;			
		ELSIF nEvent = E_SM_EVENT.READ THEN
			nReadType	:= E_RS_BASE_READ_TYPE.SINGLE;
			ActivityMonitoring(FALSE);	// Reset Monitoring method
			SetState(E_RS_BASE_STATE.OP, E_RS_BASE_SUBSTATE.OP_MONITORING);
			RETURN;			
		ELSIF nEvent = E_SM_EVENT.READ_USER THEN
			nReadType	:= E_RS_BASE_READ_TYPE.SINGLE_USER;
			ActivityMonitoringUser(FALSE);	// Reset Monitoring method
			SetState(E_RS_BASE_STATE.OP, E_RS_BASE_SUBSTATE.OP_MONITORING_USER);
			RETURN;			
		ELSIF nEvent = E_SM_EVENT.MONITOR OR nEvent = E_SM_EVENT.ENABLE THEN
			nReadType	:= E_RS_BASE_READ_TYPE.PERIODIC;
			ActivityMonitoring(FALSE);	// Reset Monitoring method
			SetState(E_RS_BASE_STATE.OP, E_RS_BASE_SUBSTATE.OP_MONITORING);
			RETURN;			
		ELSIF nEvent = E_SM_EVENT.MONITOR_USER THEN
			nReadType	:= E_RS_BASE_READ_TYPE.PERIODIC_USER;
			ActivityMonitoringUser(FALSE);	// Reset Monitoring method
			SetState(E_RS_BASE_STATE.OP, E_RS_BASE_SUBSTATE.OP_MONITORING_USER);
			RETURN;			
		END_IF
		
	END_CASE
	
	// Transitions from OP state.
	// Valid for any OP substate.
	IF nEvent = E_SM_EVENT.ERRHW THEN
		ActionUnexpExecute();
		SetState(E_RS_BASE_STATE.OP, E_RS_BASE_SUBSTATE.OP_ERROR);
		RETURN;
	ELSIF nEvent = E_SM_EVENT.ERRCOMM THEN
		SetState(E_RS_BASE_STATE.OP, E_RS_BASE_SUBSTATE.OP_ERROR);
		RETURN;
	END_IF
	
END_CASE

(* 
	"Global" internal transitions valid in any state should go here.
	They do not change the active state configuration. 
	They are evaluated after all the others transitions have been 
	considered.
*) 
IF nEvent = E_SM_EVENT.RESET THEN
	ActionResetExecute();
	SetState(E_RS_BASE_STATE.NOTOP, E_RS_BASE_SUBSTATE.NOTOP_NOTREADY);
	RETURN;
END_IF
END_METHOD

END_FUNCTION_BLOCK

// POUs/Coolers/FB_RS_COMM_CRYOTELGT
FUNCTION_BLOCK FB_RS_COMM_CRYOTELGT EXTENDS FB_RS_COMM_BASE
VAR_INPUT
END_VAR
VAR_OUTPUT
END_VAR
VAR CONSTANT
END_VAR
VAR
	{attribute 'OPC.UA.DA' := '1'}
	cfg:		T_RS_COMM_CFG;				// Config parameters
	{attribute 'OPC.UA.DA' := '1'}
	ctrl:		T_RS_COMM_CTRL;				// Control parameters
	{attribute 'OPC.UA.DA' := '1'}
	{attribute 'OPC.UA.DA.Access' := '1'}
	info:		T_RS_COMM_INFO; 			// Info parameters - ReadOnly
	{attribute 'OPC.UA.DA' := '1'}
	{attribute 'OPC.UA.DA.Access' := '1'}
	stat:		T_RS_COMM_STAT;				// Status parameters - ReadOnly

	sim:		FB_SIM_RS_COMM_CRYOTELGT;		// COMM simulator

	// Physical signals - to be mapped to EL60xx serial port controller !!!
	COMin_EL60xx	AT %I* 	: KL6inData22B;	(* linked to the EL60xx *)
	COMout_EL60xx	AT %Q*	: KL6outData22B;(* linked to the EL60xx *)

	(* Serial line control *)
	COMportControl: 		SerialLineControl;

END_VAR

// Set references
cfgRef	REF=cfg;
ctrlRef	REF=ctrl;
infoRef	REF=info;
statRef	REF=stat;
simRef	REF=sim;

SUPER^();

METHOD M_ActionInitExecute
VAR_INPUT
END_VAR
//
// Copy input parameters to cfg
//
cfg.sCmdSuffix		:= in_sCmdSuffix;
cfg.sReplySuffix	:= in_sReplySuffix;
cfg.nTimeout		:= in_nTimeout;

//
// If in simulation, there is no need to reset anything.
// Just set it to initialised and go to IDLE state.
//
IF in_bSimulation THEN
	fbTimer (IN := FALSE);
	statRef.bInitialised	:= TRUE;
	statRef.nStatus			:= E_RS_COMM_STATUS.IDLE;
	statRef.sStatus			:= 'INITIALISED';
	State 					:= E_RS_COMM_STATE.IDLE;
ELSE
	stat.bInitialised	:= FALSE;
	stat.sStatus		:= 'INITIALISING';
	stat.nStatus		:= E_RS_COMM_STATUS.BUSY;
	stat.sReply 		:= ''; (* No reply yet *)
	stat.nErrorCode		:= E_RS_COMM_ERROR.OK;
	stat.sErrorText		:= 'OK';
	
	// Reset the connected serial hardware 
	ComReset (
		Execute 	:= FALSE,
		pComIn		:= ADR(COMin_EL60xx),
		pComOut		:= ADR(COMout_EL60xx),
		SizeComIn	:= SIZEOF(COMin_EL60xx),
		);
	
	// Set next state
	State 	:= E_RS_COMM_STATE.RESET;
END_IF
END_METHOD

METHOD M_ComPortControl
VAR_INPUT
END_VAR
// RS specific call of the background communication process
COMportControl(
	Mode		:= ComSerialLineMode_t.SERIALLINEMODE_KL6_22B_STANDARD,
	pComIn		:= ADR(COMin_EL60xx),					(* I/O data; see global variables *)
	pComOut		:= ADR(COMout_EL60xx),					(* I/O data; see global variables *)
	SizeComIn	:= UINT_TO_INT(SIZEOF(COMin_EL60xx)),	(* I/O data; see global variables *)
	TxBuffer	:= TxBuffer,							(* transmit buffer; see global variables *)
	RxBuffer	:= RxBuffer);							(* receive buffer; see global variables *)
END_METHOD

METHOD M_Reset
VAR_INPUT
END_VAR
// RS specific call of communication reset
//
// Reset the connected serial hardware.
ComReset (
	Execute 	:= TRUE,
	pComIn		:= ADR(COMin_EL60xx),
	pComOut		:= ADR(COMout_EL60xx),
	SizeComIn	:= SIZEOF(COMin_EL60xx),
	);

(* Next step is to clear the buffers *)
IF ComReset.Done THEN
	fbTimer (IN := FALSE);	// Reset the timer
	State 		:= E_RS_COMM_STATE.CLEAR_BUFFER;
END_IF
END_METHOD

END_FUNCTION_BLOCK

// POUs/Coolers/FB_SIM_RS_COMM_CRYOTELGT
FUNCTION_BLOCK FB_SIM_RS_COMM_CRYOTELGT EXTENDS FB_SIM_RS_COMM_BASE
VAR_INPUT
END_VAR
VAR_OUTPUT
END_VAR
VAR
	//
	// Status structure for Cryotel GT devices
	//
	// Status attributes that are read from the controller via RS-232
	sVersion:			STRING	:= 'v1.5.3 SIM';
	sMode:				STRING	:= 'GT';
	sSensor:			STRING	:= 'PT-100';
	sCtrlError:			STRING	:= '00000000';
	sCtrlMode:			STRING	:= 'OFF';
	
	lrPowerMeasured:	LREAL	:= 0.0;
	lrPowerCommanded:	LREAL	:= 240.0;
	lrTempColdHead:		LREAL	:= 289.15;	// Room temperature (289.15K = 16.0C) to start with.
	lrTempReject:		LREAL	:= 25.3;	// [C]
	lrTempTarget:		LREAL	:= 0.0;		// Not used
	
	
	fbTimer:		TON;

END_VAR

M_ActivityDo();	// Implement ramps, if any

SUPER^();

METHOD M_ActivityDo
VAR_INPUT
END_VAR
VAR
	lrProgress:	LREAL;
END_VAR
fbTimer();

IF sCtrlMode = 'POWER' THEN
	IF NOT fbTimer.Q	THEN
		lrProgress		:= TIME_TO_LREAL(fbTimer.ET) / TIME_TO_LREAL(fbTimer.PT);
		lrTempColdHead	:= 	289.15 - (289.15 - 80.0) * lrProgress;
	ELSE
		lrTempColdHead	:= 80.0;
	END_IF
END_IF
END_METHOD

METHOD M_GetSimReply : STRING(255)
VAR_INPUT
	{attribute 'OPC.UA.DA' := '0'}
	in_sReceived:	STRING(255);		// String received from a client
END_VAR
VAR
	sReply:	STRING(255);
	sTempStr:	STRING;
	lrVal:	LREAL;
	i:		INT;
    fbFormat   : FB_FormatString;
    sOut       : T_MaxString;
	nCh:	INT := 8;	// Number of channels for models 218 and 224
END_VAR
// Simulated reply has to include the echo of the command.
// For example:
//    command = 'VERSION'
//    reply   = 'VERSION$R$Nv1.5.3$R'

IF FIND (in_sReceived, 'VERSION') = 1 THEN
	sTempStr		:= CONCAT('VERSION$R$N', sVersion);
	M_GetSimReply	:= CONCAT(sTempStr,in_sReplySuffix);
ELSIF FIND (in_sReceived, 'MODE') = 1 THEN
	sTempStr		:= CONCAT('MODE$R$N', sMode);
	M_GetSimReply	:= CONCAT(sTempStr,in_sReplySuffix);
ELSIF FIND (in_sReceived, 'SENSOR') = 1 THEN
	sTempStr		:= CONCAT('SENSOR$R$N', sSensor);
	M_GetSimReply	:= CONCAT(sTempStr,in_sReplySuffix);
ELSIF FIND (in_sReceived, 'PWOUT=') = 1 THEN
	// Example:         'PWOUT=240$R'.
	// Reply should be: 'PWOUT=240$R$N240.00$R'.
	// Get the value from the command, i.e. everything after 'PWOUT='.
	sTempStr			:= MID(in_sReceived, LEN(in_sReceived)-6, 7);	// = '240$R'
	lrPowerCommanded	:= STRING_TO_LREAL(sTempStr);	// = 240.0
	sTempStr			:= CONCAT(in_sReceived, '$N');	// 'PWOUT=240$R' + '$N' = 'PWOUT=240$R$N' 
	M_GetSimReply		:= CONCAT(sTempStr, M_Get_LREAL_TO_STRING(lrPowerCommanded,2));
ELSIF FIND (in_sReceived, 'PWOUT') = 1 THEN
	M_GetSimReply	:= CONCAT('PWOUT$R$N', M_Get_LREAL_TO_STRING(lrPowerCommanded,2));
ELSIF FIND (in_sReceived, 'P') = 1 THEN
	lrPowerMeasured	:= M_GenerateRandom_LREAL(lrPowerCommanded-0.3,0.3);
	M_GetSimReply	:= CONCAT('P$R$N', M_Get_LREAL_TO_STRING(lrPowerMeasured,2));
ELSIF FIND (in_sReceived, 'ERROR') = 1 THEN
	sTempStr		:= CONCAT('ERROR$R$N', sCtrlError);
	M_GetSimReply	:= CONCAT(sTempStr,in_sReplySuffix);
ELSIF FIND (in_sReceived, 'COOLER=POWER') = 1 THEN
	sCtrlMode		:= 'POWER';
	M_GetSimReply	:= CONCAT('COOLER=POWER$R$NPOWER',in_sReplySuffix);
	// Start ramping down the cold head temperature,
	// starting fromroom temperature.
	lrTempColdHead	:= 289.15;	
	fbTimer(IN:=FALSE);
	fbTimer(IN:=TRUE, PT:=T#60S);
ELSIF FIND (in_sReceived, 'COOLER=OFF') = 1 THEN
	fbTimer(IN:=FALSE);	// Stop the temperature ramp.
	sCtrlMode			:= 'OFF';
	M_GetSimReply		:= CONCAT('COOLER=OFF$R$NOFF',in_sReplySuffix);
	lrPowerCommanded	:= 240.0;
	lrPowerMeasured		:= 0.0;
	lrTempColdHead		:= 289.15;
ELSIF FIND (in_sReceived, 'COOLER') = 1 THEN
	sTempStr		:= CONCAT('COOLER$R$N', sCtrlMode);
	M_GetSimReply	:= CONCAT(sTempStr,in_sReplySuffix);
ELSIF FIND (in_sReceived, 'TC') = 1 THEN
	M_GetSimReply	:= CONCAT('TC$R$N', M_Get_LREAL_TO_STRING(lrTempColdHead,2));
ELSIF FIND (in_sReceived, 'TEMP RJ') = 1 THEN
	// Reject temperature [C] !!! should always be close to 
	// the room temperature and slightly above the 
	// cold head temperature [K].
	// So, we have to convert K to C.
	lrTempReject	:= M_GenerateRandom_LREAL(MAX(16.0,lrTempColdHead-273.15),0.1);
	M_GetSimReply	:= CONCAT('TEMP RJ$R$N', M_Get_LREAL_TO_STRING(lrTempReject,2));
ELSE
	// Unknown command.
	// Return '<CR><LF><CR>', i.e. '$R$N$R' in order to complete the reading.
	M_GetSimReply	:= CONCAT('$R$N', in_sReplySuffix);
END_IF
END_METHOD

END_FUNCTION_BLOCK

// POUs/Pumps/FB_CRYO_PUMP_BASE
// Cryo Pump Control Base FB
FUNCTION_BLOCK FB_CRYO_PUMP_BASE EXTENDS FB_RS_BASE
VAR_INPUT
	{attribute 'OPC.UA.DA' := '0'}
	in_bEnable:			BOOL;			// Flag to Start/Stop pump
	{attribute 'OPC.UA.DA' := '0'}
	in_nModel:			DINT := 2303;	// Model number
	{attribute 'OPC.UA.DA' := '0'}
	in_bAutoMonitor:	BOOL := TRUE;	// If true, it starts PERIODIC reads (monitoring) after INIT
	{attribute 'OPC.UA.DA' := '0'}
	in_nPeriod:			DINT := 10000;	// Interval for periodic reading [ms], default 10000 ms = 10 sec
END_VAR
VAR_OUTPUT
END_VAR
VAR
	{attribute 'OPC.UA.DA' := '0'}
	cfgBaseRef:			REFERENCE TO T_CRYO_PUMP_BASE_CFG;	
	{attribute 'OPC.UA.DA' := '0'}
	ctrlBaseRef:		REFERENCE TO T_CRYO_PUMP_BASE_CTRL;	
	{attribute 'OPC.UA.DA' := '0'}
	statBaseRef:		REFERENCE TO T_CRYO_PUMP_BASE_STAT;	

	// Pointers to arrays of INIT and READ commands
	{attribute 'OPC.UA.DA' := '0'}
	ptrInitCmds:	POINTER TO ARRAY [1..8]  OF T_CRYO_PUMP_CMD;(* Pointer to INIT commands *)
	{attribute 'OPC.UA.DA' := '0'}
	ptrReadCmds:	POINTER TO ARRAY [1..16] OF T_CRYO_PUMP_CMD;(* Pointer to READ commands *)


	(* Timers *)
	{attribute 'OPC.UA.DA' := '0'}
	fbTimer:		TON; 	// General Timeout
	timerState:		TON;	// Timer for state changes
	
	// Triggers
	triggerStart:	R_TRIG;
	triggerStop:	F_TRIG;
	

	(* Misc internal vars *)
	{attribute 'OPC.UA.DA' := '0'}
	cmdCounter:		INT := 1;	// Position in commands table
	{attribute 'OPC.UA.DA' := '0'}
	bResult:		BOOL := FALSE;
	{attribute 'OPC.UA.DA' := '0'}
	bStarted:		BOOL := FALSE;

	// TODO: Add Input signals in Fbs that EXTEND this FB.

	// Output signals
	q_bStart		AT %Q*:	BOOL;	// Start/Stop the pump. Common to all.

END_VAR

// Hard-coded configuration
M_Configure();

(* Execute comm instance *)
M_ExecuteComm();
//comm(in_sCmdSuffix:=in_sCmdSuffix, in_sReplySuffix:=in_sReplySuffix, in_nTimeout:=3000);

// Update pump status from digital signals.
M_UpdateStatus();

// Capture Start/Stop commands and execute the State Machine
M_StateMachine();

// Execute the base class object FB_RS_BASE
SUPER^();

METHOD ActivityInitializing
VAR_INPUT
	bExecute:	BOOL;
END_VAR
VAR_INST
	{attribute 'OPC.UA.DA' := '0'}
    nMethodState:	INT := 0;	// State Machine current state
END_VAR
END_METHOD

METHOD ActivityMonitoring
VAR_INPUT
	bExecute:	BOOL;
END_VAR
VAR_INST
	{attribute 'OPC.UA.DA' := '0'}
    nMethodState:	INT := 0;	// State Machine current state
	{attribute 'OPC.UA.DA' := '0'}
	nRetries:		INT := 0;	// Number of retries in case of communication problems
END_VAR

VAR
	offset: INT;
END_VAR
END_METHOD

METHOD CheckForEvents
VAR_INPUT
END_VAR
VAR
END_VAR

(* 
	Start assuming the HW is OK in case there was no communication problem. 
	This is needed to recover from the situation where 
	the HW was failing and now it is working.
*)

//IF NOT bCommProblem	THEN
//	nInternalEvent := E_SM_EVENT.HWOK;
//END_IF




(* 
	Check for events in the following order: 
   	1) HW failure: without HW avilability there is no point to do anything
	2) Internal events: to allow completing the initiated commands before 
                        starting processing new commands. 
   	3) Commands: to react to external commands. Commands should be executed 
                 before processing HW signals to allow to start a recovery action.
   	4) HW signals: if any.
*)

IF NOT M_GetCouplerState() THEN	
	(* Check if the HW is NOT OK *)
	(*
	If the hardware status is NOT OK, we cannot trust the readings.
	Variable i_nCouplerState has to be mapped to a State of a terminal, e.g. EK1100.
	The value should be 8.
 	*)
	SetEvent(E_SM_EVENT.ERRHW);
	SetStatus(E_SM_ERROR.HW_NOT_OP, 'ERROR: HW not in OPERATIONAL state');
	
ELSIF M_GetCouplerState() AND statRef.nErrorCode = E_SM_ERROR.HW_NOT_OP THEN
	SetEvent(E_SM_EVENT.HWOK);

ELSIF ctrlRef.bExecute  THEN
	(* Handle commands *)
	ctrlRef.bExecute		:= FALSE;			(* Clear the Execute bit *)
	SetLastCommand(ctrlRef.nCommand);			(* Save the last command *)
	SetEvent(ctrlRef.nCommand);
	ctrlRef.nCommand 	:= E_RS_COMMAND.NONE;	(* Clear the Command *)
ELSIF nInternalEvent <> E_SM_EVENT.NONE THEN
	(* Handle internal events *)
	SetEvent(nInternalEvent);
	nInternalEvent := E_SM_EVENT.NONE;
ELSE
	(* Handle HW problems and unexpected bahaviour *)
	
END_IF
END_METHOD

METHOD M_Configure
VAR_INPUT
END_VAR
VAR
	
END_VAR
// TODO: Implement specific configuration
END_METHOD

METHOD M_ExecuteComm
VAR_INPUT
END_VAR
END_METHOD

METHOD M_GetCouplerState : BOOL
VAR_INPUT
END_VAR
END_METHOD

METHOD M_GetSpeed : DINT
VAR_INPUT
END_VAR
END_METHOD

METHOD M_IsReady : BOOL
VAR_INPUT
END_VAR
END_METHOD

METHOD M_IsRunning : BOOL
VAR_INPUT
END_VAR
END_METHOD

METHOD M_StateMachine
VAR_INPUT
END_VAR
//////////////////////
// Pump State Machine
//////////////////////
CASE statBaseRef.nPumpState OF
	E_CRYO_PUMP_STATE.OFF:
		// Capture START command
		triggerStart(CLK:=in_bEnable);
		IF triggerStart.Q THEN
			// in_bEnable is TRUE, start the pump.
			ctrlBaseRef.bStart		:= TRUE;
			statBaseRef.nPumpState	:= 	E_CRYO_PUMP_STATE.STARTING;
			statBaseRef.sPumpState	:= 'Starting...';
			// Restart the timer
			timerState(IN:=FALSE);
			timerState(IN:=TRUE,PT:=UDINT_TO_TIME(cfgBaseRef.nTimeoutState));
		END_IF
	E_CRYO_PUMP_STATE.STARTING:
		timerState();
		triggerStop(CLK:= in_bEnable);
		IF timerState.Q THEN
			// Timeout, stop the pump.
			ctrlBaseRef.bStart		:= FALSE;
			timerState(IN:=FALSE);
			statBaseRef.nPumpState	:= 	E_CRYO_PUMP_STATE.ERROR;
			statBaseRef.sPumpState	:= 'ERROR - Timeout on START';
		ELSIF M_IsReady() THEN
			timerState(IN:=FALSE);
			statBaseRef.nPumpState	:= 	E_CRYO_PUMP_STATE.ON;
			statBaseRef.sPumpState	:= 'ON';
		ELSIF triggerStop.Q THEN
			// in_bEnable is FALSE, stop the pump.
			ctrlBaseRef.bStart		:= FALSE;
			// Restart the timer
			timerState(IN:=FALSE);
			timerState(IN:=TRUE,PT:=UDINT_TO_TIME(cfgBaseRef.nTimeoutState));
			statBaseRef.nPumpState	:= 	E_CRYO_PUMP_STATE.STOPPING;
			statBaseRef.sPumpState	:= 'Stopping...';
		END_IF
	E_CRYO_PUMP_STATE.ON:
		triggerStop(CLK:= in_bEnable);
		IF triggerStop.Q THEN
			// in_bEnable is FALSE, stop the pump.
			// Restart the timer
			ctrlBaseRef.bStart		:= FALSE;
			timerState(IN:=FALSE);
			timerState(IN:=TRUE,PT:=UDINT_TO_TIME(cfgBaseRef.nTimeoutState));
			statBaseRef.nPumpState	:= 	E_CRYO_PUMP_STATE.STOPPING;
			statBaseRef.sPumpState	:= 'Stopping...';
		ELSIF NOT M_IsReady()  OR  NOT M_IsRunning() THEN
			ctrlBaseRef.bStart		:= FALSE;
			statBaseRef.nPumpState	:= 	E_CRYO_PUMP_STATE.ERROR;
			statBaseRef.sPumpState	:= 'ERROR - Unexpected STOP';
		END_IF
	E_CRYO_PUMP_STATE.STOPPING:
		timerState();
		// Capture START command
		triggerStart(CLK:=in_bEnable);
		IF timerState.Q THEN
			timerState(IN:=FALSE);
			statBaseRef.nPumpState	:= 	E_CRYO_PUMP_STATE.ERROR;
			statBaseRef.sPumpState	:= 'ERROR - Timeout on STOP';
		ELSIF NOT M_IsReady()  AND NOT M_IsRunning() THEN
			timerState(IN:=FALSE);
			statBaseRef.nPumpState	:= 	E_CRYO_PUMP_STATE.OFF;
			statBaseRef.sPumpState	:= 'OFF';
		ELSIF triggerStart.Q THEN
			// in_bEnable is TRUE, start the pump.
			ctrlBaseRef.bStart		:= TRUE;
			statBaseRef.nPumpState	:= 	E_CRYO_PUMP_STATE.STARTING;
			statBaseRef.sPumpState	:= 'Starting...';
			// Restart the timer
			timerState(IN:=FALSE);
			timerState(IN:=TRUE,PT:=UDINT_TO_TIME(cfgBaseRef.nTimeoutState));
		END_IF
	E_CRYO_PUMP_STATE.ERROR:
		// To recover from error, STOP command has to be issued
		// in order to reset triggerStop.
		// Capture STOP command
		triggerStop(CLK:=in_bEnable);
		IF triggerStop.Q THEN
			// in_bEnable is TRUE, start the pump.
			statBaseRef.nPumpState	:= 	E_CRYO_PUMP_STATE.OFF;
			statBaseRef.sPumpState	:= 'OFF';
		END_IF
		
		// If in_bEnable is FALSE, Capture START command.
		triggerStart(CLK:=in_bEnable);
		IF triggerStart.Q THEN
			// in_bEnable is TRUE, start the pump.
			ctrlBaseRef.bStart		:= TRUE;
			statBaseRef.nPumpState	:= 	E_CRYO_PUMP_STATE.STARTING;
			statBaseRef.sPumpState	:= 'Starting...';
			// Restart the timer
			timerState(IN:=FALSE);
			timerState(IN:=TRUE,PT:=UDINT_TO_TIME(cfgBaseRef.nTimeoutState));
		END_IF
END_CASE


// Update outputs
q_bStart	:= ctrlBaseRef.bStart;
END_METHOD

METHOD M_UpdateStatus
VAR_INPUT
END_VAR
// TODO: For each pump FB that extends FB_CRYO_PUMP_BASE update inputs in M_UpdateStatus(), e.g.

(*
// Update inputs
stat.bReady		:= i_bReady;
stat.bSpeed100	:= i_bSpeed100;
stat.bWarning	:= i_bWarning;
stat.bAlarm		:= i_bAlarm;

CASE stat.nCtrlMode	OF
	0:	stat.sCtrlMode	:= 'HHR (Hand-Held Remote)';
	1:	stat.sCtrlMode	:= 'REMOTE';
	2:	stat.sCtrlMode	:= 'SERIAL LINK';
	3:	stat.sCtrlMode	:= 'FIELDBUS';
ELSE
	stat.sCtrlMode	:= 'UNKNOWN';
END_CASE

*)
END_METHOD

METHOD ProcessEvents
VAR_INPUT
END_VAR

(* 
	Before processing the event, execute the Do-Activity tasks. 
	Note that, in case of orthogonal regions, more than one Do-Activity 
	could run in the same PLC cycle.
	Note: Most of these activities have timeouts since they take time.
*)

IF	statRef.nSubstate = E_RS_BASE_SUBSTATE.OP_MONITORING 		OR 
	statRef.nSubstate = E_RS_BASE_SUBSTATE.NOTOP_READY			OR
	(statRef.nSubstate = E_RS_BASE_SUBSTATE.NOTOP_ERROR 	AND 
	 nLastGoodSubstate = E_RS_BASE_SUBSTATE.NOTOP_READY) 		OR 
	(statRef.nSubstate = E_RS_BASE_SUBSTATE.OP_ERROR 		AND 
	 nLastGoodSubstate = E_RS_BASE_SUBSTATE.OP_MONITORING)			THEN
	ActivityMonitoring(TRUE);
ELSIF statRef.nSubstate = E_RS_BASE_SUBSTATE.OP_MONITORING_USER THEN
	ActivityMonitoringUser(TRUE);
ELSIF statRef.nSubstate = E_RS_BASE_SUBSTATE.NOTOP_INITIALIZING THEN
	ActivityInitializing(TRUE);
END_IF

// Set last known good substate. Used for recovery from comm problems.
M_SetLastGoodSubstate();

(* 
	Evaluate state machine transitions.
*)

CASE statRef.nState OF

//***********************************
// NOTOP
//***********************************
E_RS_BASE_STATE.NOTOP:

	(* Transitions from NOTOP substates *)
	CASE statRef.nSubstate OF
	
	E_RS_BASE_SUBSTATE.NOTOP_NOTREADY:		
		IF 	nEvent = E_SM_EVENT.INIT OR cfgRef.bAutoMonitor  THEN
			nEvent := E_SM_EVENT.INIT;
			ActionInitExecute();
			SetState(E_RS_BASE_STATE.NOTOP, E_RS_BASE_SUBSTATE.NOTOP_INITIALIZING);
			SetStatus(E_SM_ERROR.OK, 'OK');
			RETURN;
		END_IF
		
	E_RS_BASE_SUBSTATE.NOTOP_INITIALIZING:			
		IF nEvent = E_SM_EVENT.INITDONE THEN
			nReadType := E_RS_BASE_READ_TYPE.PERIODIC;
			ActivityMonitoring(FALSE);	// Reset Monitoring method
			IF cfgRef.bAutoMonitor THEN
				nEvent := E_SM_EVENT.ENABLE;
				statRef.bAutoStarted	:= TRUE;
				SetState(E_RS_BASE_STATE.OP, E_RS_BASE_SUBSTATE.OP_MONITORING);
			ELSE
				SetState(E_RS_BASE_STATE.NOTOP, E_RS_BASE_SUBSTATE.NOTOP_READY);
			END_IF
			RETURN;
		ELSIF nEvent = E_SM_EVENT.ERRINIT THEN
			// INIT failed. Keep re-trying.
			SetState(E_RS_BASE_STATE.NOTOP, E_RS_BASE_SUBSTATE.NOTOP_NOTREADY);
			RETURN;
		END_IF
		
	E_RS_BASE_SUBSTATE.NOTOP_READY:			
		IF nEvent = E_SM_EVENT.ENABLE THEN
			IF cfgRef.bAutoMonitor THEN
				// Monitoring is already in progress.
				// It has to complete the read cycle in a clean way.
				nNextState		:= E_RS_BASE_STATE.OP;					// Next state after STOP	
				nNextSubstate	:= E_RS_BASE_SUBSTATE.OP_MONITORING;	// Next substate after STOP	
				nNextDescription:= 'BUSY';
				nReadType		:= E_RS_BASE_READ_TYPE.PERIODIC;
				RETURN;
			ELSE
				SetState(E_RS_BASE_STATE.OP, E_RS_BASE_SUBSTATE.OP_MONITORING);
				// This call MUST be after SetState()
				ActivityMonitoring(FALSE);	// Reset Monitoring method
			END_IF
		END_IF

	E_RS_BASE_SUBSTATE.NOTOP_ERROR:			
		IF nEvent = E_SM_EVENT.HWOK THEN
			SetState(E_RS_BASE_STATE.NOTOP, E_RS_BASE_SUBSTATE.NOTOP_NOTREADY);
			RETURN;
		ELSIF nEvent = E_SM_EVENT.COMMOK THEN
			SetState(E_RS_BASE_STATE.NOTOP, nLastGoodSubstate);
			RETURN;			
		END_IF
		
	END_CASE

	(* Transitions from NOTOP state *)
	IF	nEvent = E_SM_EVENT.ERRHW OR
		nEvent = E_SM_EVENT.ERRCOMM	THEN
		ActionUnexpExecute();
		SetState(E_RS_BASE_STATE.NOTOP, E_RS_BASE_SUBSTATE.NOTOP_ERROR);
		RETURN;
	END_IF
	
//***********************************
// OPERATIONAL
//***********************************
E_RS_BASE_STATE.OP:

	(* Transitions from OP subastates *)
	CASE statRef.nSubstate OF
	E_RS_BASE_SUBSTATE.OP_ERROR:			
		IF nEvent = E_SM_EVENT.HWOK THEN
			SetStatus(E_SM_ERROR.OK, 'OK');
			SetState(E_RS_BASE_STATE.OP, E_RS_BASE_SUBSTATE.OP_IDLE);
			RETURN;			
		ELSIF nEvent = E_SM_EVENT.DISABLE THEN
			ActionDisableExecute();
			SetState(E_RS_BASE_STATE.NOTOP, E_RS_BASE_SUBSTATE.NOTOP_ERROR);
			RETURN;			
		ELSIF nEvent = E_SM_EVENT.COMMOK THEN
			SetState(E_RS_BASE_STATE.OP, nLastGoodSubstate);
			RETURN;			
		END_IF

	E_RS_BASE_SUBSTATE.OP_MONITORING:
		IF nEvent = E_SM_EVENT.DISABLE THEN
			ActionDisableExecute();
			RETURN;			
		ELSIF nEvent = E_SM_EVENT.STOPMON THEN
			ActionStopExecute();
			RETURN;			
		ELSIF nEvent = E_SM_EVENT.READDONE THEN
			SetState(E_RS_BASE_STATE.OP, E_RS_BASE_SUBSTATE.OP_IDLE);
			RETURN;			
		ELSIF nEvent = E_SM_EVENT.ERRCOMM THEN
			SetState(E_RS_BASE_STATE.OP, E_RS_BASE_SUBSTATE.OP_ERROR);
			RETURN;			
		END_IF
		
	E_RS_BASE_SUBSTATE.OP_MONITORING_USER:			
		IF nEvent = E_SM_EVENT.DISABLE THEN
			ActionDisableExecute();
			RETURN;			
		ELSIF nEvent = E_SM_EVENT.STOPMON THEN
			ActionStopExecute();
			RETURN;			
		ELSIF nEvent = E_SM_EVENT.READDONE THEN
			SetState(E_RS_BASE_STATE.OP, E_RS_BASE_SUBSTATE.OP_IDLE);
			RETURN;			
		END_IF
		
	E_RS_BASE_SUBSTATE.OP_IDLE:			
		IF nEvent = E_SM_EVENT.DISABLE THEN
			ActionDisableExecute();
			RETURN;			
		ELSIF nEvent = E_SM_EVENT.READ THEN
			nReadType	:= E_RS_BASE_READ_TYPE.SINGLE;
			ActivityMonitoring(FALSE);	// Reset Monitoring method
			SetState(E_RS_BASE_STATE.OP, E_RS_BASE_SUBSTATE.OP_MONITORING);
			RETURN;			
		ELSIF nEvent = E_SM_EVENT.READ_USER THEN
			nReadType	:= E_RS_BASE_READ_TYPE.SINGLE_USER;
			ActivityMonitoringUser(FALSE);	// Reset Monitoring method
			SetState(E_RS_BASE_STATE.OP, E_RS_BASE_SUBSTATE.OP_MONITORING_USER);
			RETURN;			
		ELSIF nEvent = E_SM_EVENT.MONITOR OR nEvent = E_SM_EVENT.ENABLE THEN
			nReadType	:= E_RS_BASE_READ_TYPE.PERIODIC;
			ActivityMonitoring(FALSE);	// Reset Monitoring method
			SetState(E_RS_BASE_STATE.OP, E_RS_BASE_SUBSTATE.OP_MONITORING);
			RETURN;			
		ELSIF nEvent = E_SM_EVENT.MONITOR_USER THEN
			nReadType	:= E_RS_BASE_READ_TYPE.PERIODIC_USER;
			ActivityMonitoringUser(FALSE);	// Reset Monitoring method
			SetState(E_RS_BASE_STATE.OP, E_RS_BASE_SUBSTATE.OP_MONITORING_USER);
			RETURN;			
		END_IF
		
	END_CASE
	
	// Transitions from OP state.
	// Valid for any OP substate.
	IF nEvent = E_SM_EVENT.ERRHW THEN
		ActionUnexpExecute();
		SetState(E_RS_BASE_STATE.OP, E_RS_BASE_SUBSTATE.OP_ERROR);
		RETURN;
	ELSIF nEvent = E_SM_EVENT.ERRCOMM THEN
		SetState(E_RS_BASE_STATE.OP, E_RS_BASE_SUBSTATE.OP_ERROR);
		RETURN;
	END_IF
	
END_CASE

(* 
	"Global" internal transitions valid in any state should go here.
	They do not change the active state configuration. 
	They are evaluated after all the others transitions have been 
	considered.
*) 
IF nEvent = E_SM_EVENT.RESET THEN
	ActionResetExecute();
	SetState(E_RS_BASE_STATE.NOTOP, E_RS_BASE_SUBSTATE.NOTOP_NOTREADY);
	RETURN;
END_IF
END_METHOD

END_FUNCTION_BLOCK

// POUs/Pumps/FB_CRYO_PUMP_ATH2303M
FUNCTION_BLOCK FB_CRYO_PUMP_ATH2303M EXTENDS FB_CRYO_PUMP_SERIAL
VAR_INPUT
END_VAR
VAR_OUTPUT
END_VAR
VAR
	{attribute 'OPC.UA.DA' := '1'}
	cfg:		T_CRYO_PUMP_ATM2303M_CFG;	
	{attribute 'OPC.UA.DA' := '1'}
	ctrl:		T_CRYO_PUMP_BASE_CTRL;	
	{attribute 'OPC.UA.DA' := '1'}
	{attribute 'OPC.UA.DA.Access' := '1'}
	stat:		T_CRYO_PUMP_ATM2303M_STAT;	


	// Input signals
	i_bReady		AT %I*:	BOOL;	// OK for Process, i.e. speed ≥ nominal speed
	i_bSpeed100		AT %I*:	BOOL;	// pump speed > 100 rpm
	i_bWarning		AT %I*:	BOOL;	// presence of a warning
	i_bAlarm		AT %I*:	BOOL;	// presence of an alarm

END_VAR


// Execute the base class object FB_CRYO_PUMP_SERIAL
SUPER^();

METHOD M_Configure
VAR_INPUT
END_VAR
VAR
	//
	// List of INIT commands.
	//
	cmdList_Init_ATH2303M:	ARRAY [1..8] OF T_CRYO_PUMP_CMD := [
		(cmd := cfg.C_CMD_IDN, 	length := 0),	// 29?
		(cmd := cfg.C_CMD_RDI, 	length := 0),	// 11?
		(cmd := cfg.C_CMD_VER, 	length := 92),
		(cmd := '', 		length := 0),
		(cmd := '', 		length := 0),
		(cmd := '', 		length := 0),
		(cmd := '', 		length := 0),
		(cmd := '', 		length := 0)];

	//
	//	List of READ (and WRITE) commands.
	// NOTE: Monitoring loop stops on first cmd = ''.
	//
	cmdList_Read_ATH2303M:	ARRAY [1..16] OF T_CRYO_PUMP_CMD := [
		(cmd := cfg.C_CMD_SEL, 	length := 15),
		(cmd := cfg.C_CMD_STA, 	length := 78),
		(cmd := cfg.C_CMD_LEV, 	length := 66),
		(cmd := '', 		length := 0),
		(cmd := '', 		length := 0),
		(cmd := '', 		length := 0),
		(cmd := '', 		length := 0),
		(cmd := '', 		length := 0),
		(cmd := '', 		length := 0),
		(cmd := '', 		length := 0),
		(cmd := '', 		length := 0),
		(cmd := '', 		length := 0),
		(cmd := '', 		length := 0),
		(cmd := '', 		length := 0),
		(cmd := '', 		length := 0),
		(cmd := '', 		length := 0)];
	
END_VAR
IF NOT bStarted	THEN
	//
	// START: Mandatory for ALL pumps !!!
	//
	// Set references from FB_RS_BASE
	cfgRef	REF=cfg;
	ctrlRef	REF=ctrl;
	statRef	REF=stat;

	// Set references from FB_CRYO_TMP_BASE
	cfgBaseRef	REF=cfg;
	ctrlBaseRef	REF=ctrl;
	statBaseRef	REF=stat;

	// Copy input parameters to configuration
	cfg.nModel			:= in_nModel;
	cfg.bAutoMonitor	:= in_bAutoMonitor;
	cfg.tDelay_Periodic	:= DINT_TO_TIME(in_nPeriod);
	
	
	// Set pointers to arrays of commands
	ptrInitCmds	:= ADR(cfg.cmdList_Init);(* Pointer to INIT commands *)
	ptrReadCmds	:= ADR(cfg.cmdList_Read);(* Pointer to READ commands *)
	
	// TODO in FB that extends the functionality
	// Set pointers to comm, i.e.
	ptrCommCfg	:= ADR(comm.cfg);	(* Pointer to comm.cfg instance *)
	ptrCommCtrl	:= ADR(comm.ctrl);	(* Pointer to comm.ctrl instance *)
	ptrCommStat	:= ADR(comm.stat);	(* Pointer to comm.stat instance *)
	
	// Set comm suffixes for commands and replies
	ptrCommCfg^.sCmdSuffix		:= in_sCmdSuffix;
	ptrCommCfg^.sReplySuffix	:= in_sReplySuffix;

	statRef.bConfigured	:= TRUE;
	bStarted			:= TRUE;
	//
	// END: Mandatory for ALL pumps !!!
	//


	//
	// ATH specific configuration
	//
	
	// Assign INIT and READ commands.
	cfg.cmdList_Init	:= cmdList_Init_ATH2303M;
	cfg.cmdList_Read	:= cmdList_Read_ATH2303M;
END_IF
END_METHOD

METHOD M_GetSpeed : DINT
VAR_INPUT
END_VAR
M_GetSpeed	:= stat.nPumpSpeed;
END_METHOD

METHOD M_IsReady : BOOL
VAR_INPUT
END_VAR
M_IsReady	:= stat.bReady;
END_METHOD

METHOD M_IsRunning : BOOL
VAR_INPUT
END_VAR
M_IsRunning	:= stat.bMoving;
END_METHOD

METHOD M_ReadFromReply : BOOL
// Method to check correctness of the reply and assign the result to a status variable.
VAR_INPUT
	idx:		INT;		(* arr [idx] will hold the first extracted value, arr [idx+1] the second one, etc. *)
	bInitCmd:	BOOL := FALSE;
END_VAR
VAR
	pos:	INT;
	cmd:	STRING;
	length:	DINT;
	subStr:	STRING(255);
END_VAR
// During INIT it might happen that the command index is 0.
// These cases should be discarded.
IF idx <= 0	THEN
	M_ReadFromReply	:= TRUE;
	RETURN;
END_IF

IF bInitCmd	THEN
	cmd		:= cfg.cmdList_Init[idx].cmd;
	length	:= cfg.cmdList_Init[idx].length;
ELSE
	cmd		:= cfg.cmdList_Read[idx].cmd;
	length	:= cfg.cmdList_Read[idx].length;
END_IF

IF length <> 0  AND  LEN(stat.sReply) <> length THEN
	M_ReadFromReply	:= FALSE;
	RETURN;
END_IF

IF cmd = cfg.C_CMD_STA	THEN
	stat.nPumpSpeed		:= STRING_TO_DINT(MID(stat.sReply,5,10));
	stat.nMotorVolt		:= STRING_TO_DINT(MID(stat.sReply,2,36));
	stat.nMotorCurr		:= STRING_TO_DINT(MID(stat.sReply,5,39));
	stat.nPumpTemp		:= STRING_TO_DINT(MID(stat.sReply,3,45));
	stat.nElecTemp	:= STRING_TO_DINT(MID(stat.sReply,3,49));
ELSIF cmd = cfg.C_CMD_LEV	THEN
	stat.nNominalSpeed				:= STRING_TO_DINT(MID(stat.sReply,5,6));
	stat.nStandbySpeed				:= STRING_TO_DINT(MID(stat.sReply,5,12));
	stat.nPumpHours					:= STRING_TO_DINT(MID(stat.sReply,5,26));
	stat.nElecHours					:= STRING_TO_DINT(MID(stat.sReply,5,32));
	stat.nSetPoint_AtSpeed			:= STRING_TO_DINT(MID(stat.sReply,2,54));
	stat.nSetPoint_Temp				:= STRING_TO_DINT(MID(stat.sReply,2,57));
	stat.nSetPoint_BearingWarn		:= STRING_TO_DINT(MID(stat.sReply,2,60));
	stat.nSetPoint_BearingCounter	:= STRING_TO_DINT(MID(stat.sReply,3,63));
ELSIF cmd = cfg.C_CMD_IDN	THEN
	stat.sIDN	:= MID(stat.sReply, LEN(stat.sReply)-6, 6);	// Strip the string off prefix and sufix.
ELSIF cmd = cfg.C_CMD_RDI	THEN
	stat.sRDI	:= MID(stat.sReply, LEN(stat.sReply)-6, 6);	// Strip the string off prefix and sufix.
ELSIF cmd = cfg.C_CMD_VER	THEN
	subStr		:= MID(stat.sReply, LEN(stat.sReply)-6, 6);	// Strip the string off prefix and sufix.
	pos			:= FIND(subStr, ',');	// Find first comma
	stat.sVer1	:= MID(subStr, pos-1, 1);	// Assign substring up to the first comma char
	subStr		:= MID(subStr, LEN(subStr)-pos, pos+1);	// Take the string after sVer1 and comma.
	pos			:= FIND(subStr, ',');	// Find next comma
	stat.sVer2	:= MID(subStr, pos-1, 1);	// Take the string up to the comma
	subStr		:= MID(subStr, LEN(subStr)-pos, pos+1);	// Take the string after sVer1 and comma.
	pos			:= FIND(subStr, ',');	// Find next comma
	stat.sVer3	:= MID(subStr, pos-1, 1);	// Take the string up to the comma
	subStr		:= MID(subStr, LEN(subStr)-pos, pos+1);	// Take the string after sVer1 and comma.
	stat.sVer4	:= subStr;	// Take the rest as sVer4
ELSIF cmd = cfg.C_CMD_SEL	THEN
	stat.nCtrlMode		:= STRING_TO_DINT(MID(stat.sReply,1,14));
END_IF


M_ReadFromReply	:= true;	// OK
END_METHOD

METHOD M_UpdateStatus
VAR_INPUT
END_VAR
// Update Status from digital inputs readings
stat.bReady		:= i_bReady;
stat.bSpeed100	:= i_bSpeed100;
stat.bWarning	:= NOT i_bWarning;	// Active low
stat.bAlarm		:= NOT i_bAlarm;	// Active low

stat.bMoving	:= stat.bReady OR stat.bSpeed100 OR stat.nPumpSpeed > 0;

